MODBUS_INEPRO_RegAddress[i,4]:=16#2020;
MODBUS_INEPRO_RegDescr[i,4]:='Grid frequency';
MODBUS_INEPRO_RegQuantity[i,4]:=2;
MODBUS_INEPRO_RegValueType[i,4]:=VALUE_REAL;

MODBUS_INEPRO_RegAddress[i,5]:=16#2068;
MODBUS_INEPRO_RegDescr[i,5]:='L1 CURRENT';
MODBUS_INEPRO_RegQuantity[i,5]:=2;
MODBUS_INEPRO_RegValueType[i,5]:=VALUE_REAL;

MODBUS_INEPRO_RegAddress[i,6]:=16#206C;
MODBUS_INEPRO_RegDescr[i,6]:='L2 CURRENT';
MODBUS_INEPRO_RegQuantity[i,6]:=2;
MODBUS_INEPRO_RegValueType[i,6]:=VALUE_REAL;

MODBUS_INEPRO_RegAddress[i,7]:=16#2070;
MODBUS_INEPRO_RegDescr[i,7]:='L3 CURRENT';
MODBUS_INEPRO_RegQuantity[i,7]:=2;
MODBUS_INEPRO_RegValueType[i,7]:=VALUE_REAL;

MODBUS_INEPRO_RegAddress[i,8]:=16#2080;
MODBUS_INEPRO_RegDescr[i,8]:='ACTIVE POWER';
MODBUS_INEPRO_RegQuantity[i,8]:=2;
MODBUS_INEPRO_RegValueType[i,8]:=VALUE_REAL;

MODBUS_INEPRO_RegAddress[i,9]:=16#2088;
MODBUS_INEPRO_RegDescr[i,9]:='L1 ACTIVE POWER';
MODBUS_INEPRO_RegQuantity[i,9]:=2;
MODBUS_INEPRO_RegValueType[i,9]:=VALUE_REAL;

MODBUS_INEPRO_RegAddress[i,10]:=16#208C;
MODBUS_INEPRO_RegDescr[i,10]:='L2 ACTIVE POWER';
MODBUS_INEPRO_RegQuantity[i,10]:=2;
MODBUS_INEPRO_RegValueType[i,10]:=VALUE_REAL;

MODBUS_INEPRO_RegAddress[i,11]:=16#2090;
MODBUS_INEPRO_RegDescr[i,11]:='L3 ACTIVE POWER';
MODBUS_INEPRO_RegQuantity[i,11]:=2;
MODBUS_INEPRO_RegValueType[i,11]:=VALUE_REAL;

MODBUS_INEPRO_RegAddress[i,12]:=16#20A0;
MODBUS_INEPRO_RegDescr[i,12]:='REACTIVE POWER';
MODBUS_INEPRO_RegQuantity[i,12]:=2;
MODBUS_INEPRO_RegValueType[i,12]:=VALUE_REAL;

MODBUS_INEPRO_RegAddress[i,13]:=16#20A8;
MODBUS_INEPRO_RegDescr[i,13]:='L1 REACTIVE POWER';
MODBUS_INEPRO_RegQuantity[i,13]:=2;
MODBUS_INEPRO_RegValueType[i,13]:=VALUE_REAL;

MODBUS_INEPRO_RegAddress[i,14]:=16#20AC;
MODBUS_INEPRO_RegDescr[i,14]:='L2 REACTIVE POWER';
MODBUS_INEPRO_RegQuantity[i,14]:=2;
MODBUS_INEPRO_RegValueType[i,14]:=VALUE_REAL;

MODBUS_INEPRO_RegAddress[i,15]:=16#20B0;
MODBUS_INEPRO_RegDescr[i,15]:='L3 REACTIVE POWER';
MODBUS_INEPRO_RegQuantity[i,15]:=2;
MODBUS_INEPRO_RegValueType[i,15]:=VALUE_REAL;

MODBUS_INEPRO_RegAddress[i,16]:=16#20C0;
MODBUS_INEPRO_RegDescr[i,16]:='APPARENT POWER';
MODBUS_INEPRO_RegQuantity[i,16]:=2;
MODBUS_INEPRO_RegValueType[i,16]:=VALUE_REAL;

MODBUS_INEPRO_RegAddress[i,17]:=16#20C8;
MODBUS_INEPRO_RegDescr[i,17]:='L1 APPARENT POWER';
MODBUS_INEPRO_RegQuantity[i,17]:=2;
MODBUS_INEPRO_RegValueType[i,17]:=VALUE_REAL;

MODBUS_INEPRO_RegAddress[i,18]:=16#20CC;
MODBUS_INEPRO_RegDescr[i,18]:='L2 APPARENT POWER';
MODBUS_INEPRO_RegQuantity[i,18]:=2;
MODBUS_INEPRO_RegValueType[i,18]:=VALUE_REAL;

MODBUS_INEPRO_RegAddress[i,19]:=16#20D0;
MODBUS_INEPRO_RegDescr[i,19]:='L3 APPARENT POWER';
MODBUS_INEPRO_RegQuantity[i,19]:=2;
MODBUS_INEPRO_RegValueType[i,19]:=VALUE_REAL;

MODBUS_INEPRO_RegAddress[i,20]:=16#20E0;
MODBUS_INEPRO_RegDescr[i,20]:='POWER FACTOR';
MODBUS_INEPRO_RegQuantity[i,20]:=2;
MODBUS_INEPRO_RegValueType[i,20]:=VALUE_REAL;

MODBUS_INEPRO_RegAddress[i,21]:=16#20E8;
MODBUS_INEPRO_RegDescr[i,21]:='L1 POWER FACTOR';
MODBUS_INEPRO_RegQuantity[i,21]:=2;
MODBUS_INEPRO_RegValueType[i,21]:=VALUE_REAL;

MODBUS_INEPRO_RegAddress[i,22]:=16#20EC;
MODBUS_INEPRO_RegDescr[i,22]:='L2 POWER FACTOR';
MODBUS_INEPRO_RegQuantity[i,22]:=2;
MODBUS_INEPRO_RegValueType[i,22]:=VALUE_REAL;

MODBUS_INEPRO_RegAddress[i,23]:=16#20F0;
MODBUS_INEPRO_RegDescr[i,23]:='L3 POWER FACTOR';
MODBUS_INEPRO_RegQuantity[i,23]:=2;
MODBUS_INEPRO_RegValueType[i,23]:=VALUE_REAL;

MODBUS_INEPRO_RegAddress[i,24]:=16#3000;
MODBUS_INEPRO_RegDescr[i,24]:='TOTAL ACTIVE ENERGY';
MODBUS_INEPRO_RegQuantity[i,24]:=2;
MODBUS_INEPRO_RegValueType[i,24]:=VALUE_REAL;

MODBUS_INEPRO_RegAddress[i,25]:=16#3060;
MODBUS_INEPRO_RegDescr[i,25]:='TOTAL REACTIVE ENERGY';
MODBUS_INEPRO_RegQuantity[i,25]:=2;
MODBUS_INEPRO_RegValueType[i,25]:=VALUE_REAL;

MODBUS_INEPRO_RegAddress[i,26]:=16#1000;
MODBUS_INEPRO_RegDescr[i,26]:='SERIAL_NUMBER';
MODBUS_INEPRO_RegQuantity[i,26]:=2;
MODBUS_INEPRO_RegValueType[i,26]:=VALUE_LONG;

END_FOR
END_FUNCTION

(* POU Utils Functions/AVERAGE_T, ST *)
FUNCTION_BLOCK AVERAGE_T
VAR_INPUT
	IN: 	INT;
END_VAR
VAR_OUTPUT
	HI:		INT;
	AVG:	INT;
	LOW:	INT;
	ERR:	BOOL;
END_VAR
VAR
	sum:	DINT;
	cnt:	WORD;
END_VAR
IF cnt>=65000 THEN
	ERR:=TRUE;
	Read();
	sum := sum - AVG;
	cnt := cnt + 1;
END_IF

sum := sum + IN;
cnt := cnt + 1;

IF IN<LOW THEN  LOW:=IN; END_IF
IF IN>HI  THEN HI :=IN; END_IF
END_FUNCTION_BLOCK
ACTION Read:
AVG := DINT_TO_INT(sum/cnt);
END_ACTION
ACTION Reset:
HI:=IN;
AVG:=IN;
LOW:=IN;
ERR:=FALSE;

sum:=IN;
cnt:=1;
END_ACTION

(* POU ClevergyBlocks/OBJ_ANZ_INEPRO_PRO380/BUILD_REAL_COPY, ST *)
FUNCTION BUILD_REAL_COPY : REAL
VAR_INPUT
		W1	:	WORD;
		W2	:	WORD;
END_VAR
VAR
 	awWords      : ARRAY[1..2] OF WORD;
  	pReal : POINTER TO REAL;
  	rReal : REAL;
END_VAR
awWords[1] := W1;
awWords[2] := W2;
pReal := ADR(awWords);
rReal := pReal^;
BUILD_REAL_COPY:=rReal;
END_FUNCTION

(* POU Utils Functions/COPY_32SWAP16, ST *)
FUNCTION COPY_32SWAP16:BOOL
VAR_INPUT
	pSourceAddress		:POINTER TO ARRAY[1..2] OF WORD;
	pDestinationAddress	:POINTER TO ARRAY[1..2] OF WORD;
END_VAR
VAR
END_VAR
pDestinationAddress^[1]:=pSourceAddress^[2];
pDestinationAddress^[2]:=pSourceAddress^[1];
END_FUNCTION

(* POU Utils Functions/FLT_EVENT, ST *)
FUNCTION_BLOCK FLT_EVENT
VAR_INPUT
	IN		: BOOL;
	INITEV	: BOOL:=TRUE;
END_VAR
VAR_OUTPUT
	EVH		: BOOL;
	EVL		: BOOL;
END_VAR
VAR
	init	: BOOL:=FALSE;
	old		: BOOL;
END_VAR
EVH:=FALSE;
EVL:=FALSE;

IF NOT init THEN
	init:=TRUE;
	IF INITEV THEN
		old := NOT IN;
	ELSE
		old := IN;
	END_IF
END_IF

IF old<>IN THEN
	old:=IN;
	IF IN THEN EVH:=TRUE; ELSE EVL:=TRUE; END_IF
END_IF
END_FUNCTION_BLOCK

(* POU Utils Functions/FLT_TIME, ST *)
FUNCTION_BLOCK FLT_TIME
VAR_INPUT
	IN		: BOOL;
	TTAP	: TIME:=T#5s;
	INITEV	: BOOL:=TRUE;
END_VAR
VAR_OUTPUT
	OUT		: BOOL;
	EVH		: BOOL;
	EVL		: BOOL;
END_VAR
VAR
	init	: BOOL:=FALSE;
	timer	: TON;
END_VAR
EVH:=FALSE;
EVL:=FALSE;

IF NOT init THEN
	init := TRUE;
	IF INITEV THEN
		OUT  := NOT IN;
	ELSE
		OUT  := IN;
	END_IF
END_IF

IF OUT<>IN THEN
	timer(IN:=TRUE,PT:=TTAP);
	IF timer.Q THEN
		OUT:=IN;
		timer(IN:=FALSE);
		IF OUT THEN EVH:=TRUE; ELSE EVL:=TRUE; END_IF
	END_IF
ELSE
	timer(IN:=FALSE);
END_IF
END_FUNCTION_BLOCK

(* POU Utils/FUN_ByteAsci, ST *)
FUNCTION FUN_ByteAsci : STRING(1)
VAR_INPUT
	ByteIn:BYTE;
END_VAR
VAR
END_VAR
CASE ByteIn OF

	32: FUN_ByteAsci:=' ';
	33: FUN_ByteAsci:='!';
	34: FUN_ByteAsci:='"';
	35: FUN_ByteAsci:='#';

	37: FUN_ByteAsci:='%';
	38: FUN_ByteAsci:='&';

	40: FUN_ByteAsci:='(';
	41: FUN_ByteAsci:=')';
	42: FUN_ByteAsci:='*';
	43: FUN_ByteAsci:='+';
	44: FUN_ByteAsci:=',';
	45: FUN_ByteAsci:='-';
	46: FUN_ByteAsci:='.';
	47: FUN_ByteAsci:='/';
	48: FUN_ByteAsci:='0';
	49: FUN_ByteAsci:='1';
	50: FUN_ByteAsci:='2';
	51: FUN_ByteAsci:='3';
	52: FUN_ByteAsci:='4';
	53: FUN_ByteAsci:='5';
	54: FUN_ByteAsci:='6';
	55: FUN_ByteAsci:='7';
	56: FUN_ByteAsci:='8';
	57: FUN_ByteAsci:='9';
	58: FUN_ByteAsci:=':';
	59: FUN_ByteAsci:=';';
	60: FUN_ByteAsci:='<';
	61: FUN_ByteAsci:='=';
	62: FUN_ByteAsci:='>';
	63: FUN_ByteAsci:='?';
	64: FUN_ByteAsci:='@';
	65: FUN_ByteAsci:='A';
	66: FUN_ByteAsci:='B';
	67: FUN_ByteAsci:='C';
	68: FUN_ByteAsci:='D';
	69: FUN_ByteAsci:='E';
	70: FUN_ByteAsci:='F';
	71: FUN_ByteAsci:='G';
	72: FUN_ByteAsci:='H';
	73: FUN_ByteAsci:='I';
	74: FUN_ByteAsci:='J';
	75: FUN_ByteAsci:='K';
	76: FUN_ByteAsci:='L';
	77: FUN_ByteAsci:='M';
	78: FUN_ByteAsci:='N';
	79: FUN_ByteAsci:='O';
	80: FUN_ByteAsci:='P';
	81: FUN_ByteAsci:='Q';
	82: FUN_ByteAsci:='R';
	83: FUN_ByteAsci:='S';
	84: FUN_ByteAsci:='T';
	85: FUN_ByteAsci:='U';
	86: FUN_ByteAsci:='V';
	87: FUN_ByteAsci:='W';
	88: FUN_ByteAsci:='X';
	89: FUN_ByteAsci:='Y';
	90: FUN_ByteAsci:='Z';
	91: FUN_ByteAsci:='[';
	92: FUN_ByteAsci:='\';
	93: FUN_ByteAsci:=']';
	94: FUN_ByteAsci:='^';
	95: FUN_ByteAsci:='_';
	96: FUN_ByteAsci:='`';
	97: FUN_ByteAsci:='a';
	98: FUN_ByteAsci:='b';
	99: FUN_ByteAsci:='c';
	100: FUN_ByteAsci:='d';
	101: FUN_ByteAsci:='e';
	102: FUN_ByteAsci:='f';
	103: FUN_ByteAsci:='g';
	104: FUN_ByteAsci:='h';
	105: FUN_ByteAsci:='i';
	106: FUN_ByteAsci:='j';
	107: FUN_ByteAsci:='k';
	108: FUN_ByteAsci:='l';
	109: FUN_ByteAsci:='m';
	110: FUN_ByteAsci:='n';
	111: FUN_ByteAsci:='o';
	112: FUN_ByteAsci:='p';
	113: FUN_ByteAsci:='q';
	114: FUN_ByteAsci:='r';
	115: FUN_ByteAsci:='s';
	116: FUN_ByteAsci:='t';
	117: FUN_ByteAsci:='u';
	118: FUN_ByteAsci:='v';
	119: FUN_ByteAsci:='w';
	120: FUN_ByteAsci:='x';
	121: FUN_ByteAsci:='y';
	122: FUN_ByteAsci:='z';
	123: FUN_ByteAsci:='{';
	124: FUN_ByteAsci:='|';
	125: FUN_ByteAsci:='}';
	126: FUN_ByteAsci:='~';

	167: FUN_ByteAsci:='°';
	176: FUN_ByteAsci:='°';


ELSE
	FUN_ByteAsci:='';

END_CASE
END_FUNCTION

(* POU Utils Functions/LAMP_AL_GENERALE, ST *)
FUNCTION_BLOCK LAMP_AL_GENERALE
VAR_INPUT

	Allarme: BOOL;
	Warning: BOOL;
END_VAR
VAR_OUTPUT
	SistemaOK:BOOL;
	SistemaInAllarme:BOOL;
	SistemaWarning:BOOL;
	AllarmeLampada:BOOL;
END_VAR
VAR
	Lampeggio:BLINK;
END_VAR
IF Allarme THEN       					(* Se Allarme Attivo Lucde fissa ON *)
	SistemaInAllarme:=TRUE;
	SistemaWarning:=FALSE;
	AllarmeLampada:=TRUE;
ELSIF Warning THEN					(* Se Allarme Attivo Lucde fissa pulse *)
	SistemaInAllarme:=FALSE;
	SistemaWarning:=TRUE;
	Lampeggio(ENABLE:=TRUE , TIMELOW:=t#1s , TIMEHIGH:=t#1s , OUT=>AllarmeLampada );
ELSE
	SistemaInAllarme:=FALSE;
	SistemaWarning:=FALSE;
	AllarmeLampada:=FALSE;
END_IF
END_FUNCTION_BLOCK

(* POU Utils Functions/LINEAR_BAD, ST *)
FUNCTION LINEAR_BAD : INT (* Linear interpolation *)
VAR_INPUT
	PuntoMinX	: INT;
	PuntoMaxX	: INT;
	ValIn		: INT;
	PuntoMinY	: REAL;
	PuntoMaxY	: REAL;
	Decimali	: BYTE;
END_VAR
VAR
	Gain				: REAL;
	PuntoMinX_R			: REAL;
	PuntoMaxX_R			: REAL;
	Linearizzazione_R	: REAL;
END_VAR
PuntoMinX_R:=INT_TO_REAL(PuntoMinX);
PuntoMaxX_R:=INT_TO_REAL(PuntoMaxX);

Gain:=(PuntoMaxX_R-PuntoMinX_R)/(PuntoMaxY-PuntoMinY);	(* Calcolo in guadagno per la linarizzazione *)
Linearizzazione_R:=PuntoMinx+(Gain*(ValIn-PuntoMinY));	(* Ottengo il valore linearizzato *)

LINEAR_BAD:=REAL_TO_INT(Linearizzazione_R*(EXPT(10, Decimali)));  (* Ottengo intero con i decimai voluti *)
END_FUNCTION

(* POU TCP_Logger/LogTrig, ST *)
FUNCTION LogTrig : BOOL
VAR
	s1 : STRING(160);
	i  : BYTE;
	j  : WORD;
END_VAR
(*---------------------------------------------------------------*)
	Logger_Head();
(*---------------------------------------------------------------*)

PX01.AddLogData();
PX02.AddLogData();
PX03.AddLogData();
PX04.AddLogData();
Logger_Send();


Logger_Head();

(*
FOR i:=1 TO Plant_ANZ_INEPRO DO
	ANZ_INEPRO[i].AddLogData();
END_FOR *)
ANZ_INEPRO[1].AddLogData();
ANZ_INEPRO[2].AddLogData();
Logger_Send();


Logger_Head();

ANZ_INEPRO[3].AddLogData();
ANZ_INEPRO[4].AddLogData();
Logger_Send();


Logger_Head();
ANZ_INEPRO[5].AddLogData();

Logger_Send();


Logger_Head();

	COMPRESSORE01.AddLogData(ModBus:=MODB02);
	COMPRESSORE05.AddLogData(ModBus:=MODB02);
Logger_Send();


Logger_Head();
	COMPRESSORE02.AddLogData(ModBus:=MODB03);
	COMPRESSORE03.AddLogData(ModBus:=MODB03);
	COMPRESSORE04.AddLogData(ModBus:=MODB03);
Logger_Send();


Logger_Head();

	FPT01.AddLogData(ModBus:=MODB05);
	FPT02.AddLogData();
	FPT03.AddLogData();
	FPT04.AddLogData();
	FPT05.AddLogData();
	FPT06.AddLogData();
	FPT07.AddLogData();
	FPT08.AddLogData();
	FPT09.AddLogData();
	FPT10.AddLogData();

(*	ESSICATORE01.AddLogData(ModBus:=MODB04); *)
(*	ESSICATORE02.AddLogData(ModBus:=MODB04); *)



(*---------------------------------------------------------------*)
	Logger_Send();
(*---------------------------------------------------------------*)
END_FUNCTION

(* POU Utils Functions/MEMCLR, ST *)
FUNCTION MEMCLR:BOOL
VAR_INPUT
	pDestinationAddress:POINTER TO ARRAY[1..2] OF BYTE;
	BytesToClear:WORD;
END_VAR
VAR
END_VAR
WHILE (BytesToClear > 0) DO
	pDestinationAddress^[1]:=0;
	pDestinationAddress:=ADR(pDestinationAddress^[2]); (* increment destination *)
	BytesToClear:=BytesToClear -1; (* decrement number of bytes to copy *)
END_WHILE
END_FUNCTION

(* POU Plant_Objects/obj_AI_GEN, ST *)
FUNCTION_BLOCK obj_AI_GEN
(* === TEMPERATURE PROBE FROM ANALOG INPUT ===
   v1.0[16/04/05] - Versioning
*)
VAR_INPUT
	(* Settings *)
	ID				: BYTE;
	PuntoMinX		: INT;			(* Parametri per la scalatura *)
	PuntoMaxX		: INT;
	PuntoMinY		: REAL;
	PuntoMaxY		: REAL;
	Decimali		: BYTE:=1;
	SogliaHH		: WORD;			(* Soglia per segnalazione Allarme Extra Range in alto - Solitamente sondo in CC *)
	SogliaHL		: WORD;			(* Soglia per segnalazione Allarme Extra Range in Basso - Solitamente sondo Aperta *)
	SogliaWH		: REAL;			(* Soglia per segnalazione Warning  in alto  *)
	SogliaWL		: REAL;    		(* Soglia per segnalazione Warning in basso  *)
	TAP				: INT:=2000;	(* Filtro in msec *)
	INITEV			: BOOL:= TRUE;	(* Generate init OK event *)
	(* Physical input *)
	AI_INPUT		: WORD;    		(* Sensor analog input *)
	TipoSensore:STRING(12);
END_VAR
VAR_OUTPUT
	WRN				: BOOL;	(* Segnalazione Warning *)
	ERR				: BOOL; (* Segnalazione Errore *)
	ValoreScalato	: INT;
	(* Status *)
	Status_Log	: BYTE;
	Status_Vis 	: DWORD;
END_VAR
VAR
	SegnaleHH	: BOOL;
	SegnaleHL	: BOOL;
	SegnaleOK	: BOOL;
	SegnaleWH	: BOOL;
	SegnaleWL	: BOOL;
    FiltroWRN	: TON;
    FiltroOK	: TON;
    FiltroERR	: TON;
END_VAR
(* Verifico che le variabile letta dall'ingresso Analogico  sia dentro i range
ATTENZIONE I LIMITI SPESSO SONO IN WORD VERIFICA  TABELLA MANUALE WAGO  *)

SegnaleHH:=(AI_INPUT>=SogliaHH);
SegnaleHL:=(AI_INPUT<=SogliaHL);
SegnaleOK:=NOT (SegnaleHH OR SegnaleHL);

(* Linerarizzo il segnale di ingresso e la converto in unita ingegneristiche *)
ValoreScalato:=LINEAR_BAD(PuntoMinX, PuntoMaxX, AI_INPUT, PuntoMinY, PuntoMaxY, Decimali);


IF SegnaleOK  THEN
	(*  Verifica  e segnalazione Warning *)
	SegnaleWH:=(ValoreScalato>SogliaWH*(EXPT(10, Decimali)));
	SegnaleWL:=(ValoreScalato<SogliaWL*(EXPT(10, Decimali)));

	Status_Log:=0;
	Status_Vis:=16#20F020;    (* Indicazione WEB Visu Sonda OK *)

	FiltroWRN( IN:=(SegnaleWH OR SegnaleWL), PT:=INT_TO_TIME(TAP) );    (* Filtro su LOG *)
	IF  FiltroWRN.Q THEN     (* Condizione di WARNING *)
		IF NOT WRN THEN
			WRN:=TRUE;
			Status_Log:=1;
			LogEv(EL_Wrn,EO_TPV,ID,SEL(ValoreScalato<=SogliaWL,3,2),INT_TO_STRING(ValoreScalato));
		END_IF
	END_IF

    IF (INITEV OR WRN OR ERR) AND NOT FiltroWRN.Q THEN
		FiltroWRN(IN:=FALSE  , PT:=INT_TO_TIME(TAP));    (* Resetto il Filtro su LOG WRN  *)
		FiltroERR(IN:=FALSE  , PT:=INT_TO_TIME(TAP));    (* Resetto il Filtro su LOG ERR *)
		INITEV:=FALSE; ERR:=FALSE; WRN:=FALSE;
		LogEv(EL_Log,EO_TPV,ID,1,'');
	END_IF
ELSE
	FiltroERR(IN:=TRUE  , PT:= INT_TO_TIME(TAP) );    (* Filtro su LOG *)
	IF  FiltroERR.Q THEN     (* Condizione di WARNING *)
		IF NOT ERR THEN
			ERR:=TRUE;
			Status_Log:=2;

			IF SegnaleHH THEN LogEv(EL_Alarm,EO_TPV,ID,6,INT_TO_STRING(ValoreScalato));END_IF;
			IF SegnaleHL THEN LogEv(EL_Alarm,EO_TPV,ID,4,INT_TO_STRING(ValoreScalato));END_IF;
		END_IF
	END_IF

	Status_Vis:=16#2020F0;   (* Indicazione WEB Visu Sonda KO *)
END_IF



(* Status Log *)
IF ERR THEN
	Status_Log := 2;
	Status_Vis := COLOR_RED;
ELSIF WRN THEN
	Status_Log := 1;
	Status_Vis := COLOR_YELLOW;
ELSE
	Status_Log := 0; Status_Vis := COLOR_GREEN;
END_IF
END_FUNCTION_BLOCK
ACTION AddLogData:
Logger.s1:=CONCAT('&',TipoSensore);
IF ID<10 THEN Logger.s1:=CONCAT(Logger.s1,'0');END_IF
Logger.s1:=CONCAT(Logger.s1,BYTE_TO_STRING(ID));
Logger.s1:=CONCAT(Logger.s1,'=');


Logger.s1:=CONCAT(Logger.s1,WORD_TO_STRING(Status_Log));		Logger.s1:=CONCAT(Logger.s1,';');
Logger.s1:=CONCAT(Logger.s1,INT_TO_STRING(ValoreScalato));


ADDSTRING(ADR(Logger.TData), ADR(Logger.s1), Logger.TLen);
END_ACTION

(* POU ClevergyBlocks/OBJ_ANZ_INEPRO_PRO380/obj_ANZ_INEPRO_PRO380, ST *)
FUNCTION_BLOCK obj_ANZ_INEPRO_PRO380
(* === Block for realizing the ANZ entity with the meter INEPRO PRO380 ===
	
	One ANZ block manages one physical ANZ device.
	
	Versioning:
		v1.0 [28/07/16] - Diego Bernini
*)
VAR_INPUT

	(* Logical ID of the ANZ, univocal w.r.t the plant *)
	ID										 : WORD;
	(* Type of ANZ: 1-phase or 3-phase *)
	contabilizerMode							 : en_ANZ_Type := THREE_PHASE;

	modbusConnector: obj_MODBUS_GENERIC_CONNECTOR;

	(* meter dependent fields, by the connector*)
	specificData								:  typ_ANZ_INEPRO_PRO380;

	(* determines if warning errors are sent or not *)
	enableWarning : BOOL :=FALSE;

	TIMING_AGGREGATED_MEASURE:TIME;
	TIMING_RESET_AGGREGATED_MEASURE:TIME;

END_VAR

VAR_OUTPUT

	(* output records representing the data in according to the ANZ Clevergy Web format *)
	measures						: typ_ANZ_real;
	(*status of the block according the Clevergy architecture *)
	Status_Log						: BYTE;
	Status_Vis	:	DWORD;

END_VAR

VAR

	contAvg								 : REAL :=0;
	sumAvg								 : REAL :=0;
	timerCalc								 : TON;
	timerReset							 : TON;

	alarmMsg : STRING;
	alarmLaunched: ARRAY[1..MAX_ALARM] OF BYTE;

	warningMsg : STRING;
	warningLaunched: ARRAY[1..MAX_WARNING] OF BYTE;

	i : BYTE;
	tmpAlarm:BYTE;
	tmpWarning:BYTE;

END_VAR
VAR CONSTANT
	MAX_ALARM :BYTE:=20;
	MAX_WARNING :BYTE:=20;
END_VAR
VAR
	CheckEvents: BOOL;
END_VAR
Status_Log:=ModBusConnector.Status_Log;

getModbusData();

timerReset(IN:=NOT timerReset.Q,PT:=TIMING_RESET_AGGREGATED_MEASURE);
IF timerReset.Q THEN

	sumAvg := 0;
	contAvg := 0;

 	specificData.rMaximumTotalActivePower:=0; (* reset => min possible val *)
	specificData.rMaximumTotalReactivePower:= -2147483648;
	specificData.rMaximumCurrentL1:=0;
	specificData.rMaximumCurrentL2:=0;
	specificData.rMaximumCurrentL3:=0;

END_IF

(*compute additional measures, the ones which are not provided directly*)
timerCalc(IN:=NOT timerCalc.Q,PT:=TIMING_AGGREGATED_MEASURE);

IF timerCalc.Q THEN
	sumAvg := sumAvg+specificData.rTotalActivePower;
	contAvg:=contAvg+1;
	specificData.rAverageTotalActivePower:=sumAvg/contAvg;
	IF specificData.rTotalActivePower > specificData.rMaximumTotalActivePower THEN specificData.rMaximumTotalActivePower:= specificData.rTotalActivePower; END_IF
	IF specificData.rTotalReactivePower > specificData.rMaximumTotalReactivePower THEN specificData.rMaximumTotalReactivePower:= specificData.rTotalReactivePower; END_IF

	IF specificData.arCurrent[1] > specificData.rMaximumCurrentL1 THEN specificData.rMaximumCurrentL1:= specificData.arCurrent[1]; END_IF
	IF specificData.arCurrent[2] > specificData.rMaximumCurrentL2 THEN specificData.rMaximumCurrentL2:= specificData.arCurrent[2]; END_IF
	IF specificData.arCurrent[3] > specificData.rMaximumCurrentL3 THEN specificData.rMaximumCurrentL3:= specificData.arCurrent[3]; END_IF

END_IF


(* convert the data to the Clevergy format *)
convertToClevergyFormat();

(* visu	*)
IF Status_Log = 2 THEN
	Status_Vis := COLOR_RED;
ELSIF Status_Log = 1 THEN
	Status_Vis := COLOR_YELLOW;
ELSE
	Status_Vis := COLOR_GREEN;
END_IF
END_FUNCTION_BLOCK
ACTION AddLogData:
Logger.s1:=INSERT('&ANZ=',WORD_TO_STRING(ID),4);
IF ID<10 THEN Logger.s1:=INSERT(Logger.s1,'0',4); END_IF

Logger.s1:=CONCAT(Logger.s1,REAL_TO_STRING(measures.V_L1N));		Logger.s1:=CONCAT(Logger.s1,';');
Logger.s1:=CONCAT(Logger.s1,REAL_TO_STRING(measures.V_L2N));		Logger.s1:=CONCAT(Logger.s1,';');
Logger.s1:=CONCAT(Logger.s1,REAL_TO_STRING(measures.V_L3N));		Logger.s1:=CONCAT(Logger.s1,';');
Logger.s1:=CONCAT(Logger.s1,REAL_TO_STRING(measures.V_L1L2));		Logger.s1:=CONCAT(Logger.s1,';');
Logger.s1:=CONCAT(Logger.s1,REAL_TO_STRING(measures.V_L2L3));		Logger.s1:=CONCAT(Logger.s1,';');
Logger.s1:=CONCAT(Logger.s1,REAL_TO_STRING(measures.V_L3L1));		Logger.s1:=CONCAT(Logger.s1,';');

Logger.s1:=CONCAT(Logger.s1,REAL_TO_STRING(measures.FREQ));		Logger.s1:=CONCAT(Logger.s1,';');

Logger.s1:=CONCAT(Logger.s1,REAL_TO_STRING(measures.I_L1));		Logger.s1:=CONCAT(Logger.s1,';');
Logger.s1:=CONCAT(Logger.s1,REAL_TO_STRING(measures.I_L2));		Logger.s1:=CONCAT(Logger.s1,';');
Logger.s1:=CONCAT(Logger.s1,REAL_TO_STRING(measures.I_L3));		Logger.s1:=CONCAT(Logger.s1,';');
Logger.s1:=CONCAT(Logger.s1,REAL_TO_STRING(measures.I_L1_Max)); 	Logger.s1:=CONCAT(Logger.s1,';');
Logger.s1:=CONCAT(Logger.s1,REAL_TO_STRING(measures.I_L2_Max)); 	Logger.s1:=CONCAT(Logger.s1,';');
Logger.s1:=CONCAT(Logger.s1,REAL_TO_STRING(measures.I_L3_Max)); 	Logger.s1:=CONCAT(Logger.s1,';');

Logger.s1:=CONCAT(Logger.s1,REAL_TO_STRING(measures.PF_L1));		Logger.s1:=CONCAT(Logger.s1,';');
Logger.s1:=CONCAT(Logger.s1,REAL_TO_STRING(measures.PF_L2));		Logger.s1:=CONCAT(Logger.s1,';');
Logger.s1:=CONCAT(Logger.s1,REAL_TO_STRING(measures.PF_L3));		Logger.s1:=CONCAT(Logger.s1,';');

Logger.s1:=CONCAT(Logger.s1,REAL_TO_STRING(measures.P_3P));		Logger.s1:=CONCAT(Logger.s1,';');
Logger.s1:=CONCAT(Logger.s1,REAL_TO_STRING(measures.P_3P_Avg)); 	Logger.s1:=CONCAT(Logger.s1,';');
Logger.s1:=CONCAT(Logger.s1,REAL_TO_STRING(measures.P_3P_Max)); 	Logger.s1:=CONCAT(Logger.s1,';');

Logger.s1:=CONCAT(Logger.s1,REAL_TO_STRING(measures.Q_3P));			Logger.s1:=CONCAT(Logger.s1,';');
Logger.s1:=CONCAT(Logger.s1, REAL_TO_STRING(measures.Q_3P_Max));		Logger.s1:=CONCAT(Logger.s1,';');

Logger.s1:=CONCAT(Logger.s1,REAL_TO_STRING(measures.WH_3P));			Logger.s1:=CONCAT(Logger.s1,';');
Logger.s1:=CONCAT(Logger.s1,REAL_TO_STRING(measures.VARH_3P));			Logger.s1:=CONCAT(Logger.s1,';');

Logger.s1:=CONCAT(Logger.s1,BYTE_TO_STRING(Status_Log)); 					Logger.s1:=CONCAT(Logger.s1,';');

Logger.s1:=CONCAT(Logger.s1,REAL_TO_STRING(measures.COSPHI_L1));		Logger.s1:=CONCAT(Logger.s1,';');
Logger.s1:=CONCAT(Logger.s1,REAL_TO_STRING(measures.COSPHI_L2));		Logger.s1:=CONCAT(Logger.s1,';');
Logger.s1:=CONCAT(Logger.s1,REAL_TO_STRING(measures.COSPHI_L3));		Logger.s1:=CONCAT(Logger.s1,';');

Logger.s1:=CONCAT(Logger.s1,BYTE_TO_STRING(SEL(contabilizerMode=THREE_PHASE,1,0)));

ADDSTRING(ADR(Logger.TData), ADR(Logger.s1), Logger.TLen);
END_ACTION
ACTION AddLogData_OLD:
(*Logger.s1:=INSERT('&ANZ=',WORD_TO_STRING(ID),4);
IF ID<10 THEN Logger.s1:=INSERT(Logger.s1,'0',4); END_IF

Logger.s1:=CONCAT(Logger.s1,DWORD_TO_STRING(measures.V_L1N));		Logger.s1:=CONCAT(Logger.s1,';');
Logger.s1:=CONCAT(Logger.s1,DWORD_TO_STRING(measures.V_L2N));		Logger.s1:=CONCAT(Logger.s1,';');
Logger.s1:=CONCAT(Logger.s1,DWORD_TO_STRING(measures.V_L3N));		Logger.s1:=CONCAT(Logger.s1,';');
Logger.s1:=CONCAT(Logger.s1,DWORD_TO_STRING(measures.V_L1L2));		Logger.s1:=CONCAT(Logger.s1,';');
Logger.s1:=CONCAT(Logger.s1,DWORD_TO_STRING(measures.V_L2L3));		Logger.s1:=CONCAT(Logger.s1,';');
Logger.s1:=CONCAT(Logger.s1,DWORD_TO_STRING(measures.V_L3L1));		Logger.s1:=CONCAT(Logger.s1,';');

Logger.s1:=CONCAT(Logger.s1,DWORD_TO_STRING(measures.FREQ));		Logger.s1:=CONCAT(Logger.s1,';');

Logger.s1:=CONCAT(Logger.s1,DWORD_TO_STRING(measures.I_L1));		Logger.s1:=CONCAT(Logger.s1,';');
Logger.s1:=CONCAT(Logger.s1,DWORD_TO_STRING(measures.I_L2));		Logger.s1:=CONCAT(Logger.s1,';');
Logger.s1:=CONCAT(Logger.s1,DWORD_TO_STRING(measures.I_L3));		Logger.s1:=CONCAT(Logger.s1,';');
Logger.s1:=CONCAT(Logger.s1,DWORD_TO_STRING(measures.I_L1_Max)); 	Logger.s1:=CONCAT(Logger.s1,';');
Logger.s1:=CONCAT(Logger.s1,DWORD_TO_STRING(measures.I_L2_Max)); 	Logger.s1:=CONCAT(Logger.s1,';');
Logger.s1:=CONCAT(Logger.s1,DWORD_TO_STRING(measures.I_L3_Max)); 	Logger.s1:=CONCAT(Logger.s1,';');

Logger.s1:=CONCAT(Logger.s1,DINT_TO_STRING(measures.PF_L1));		Logger.s1:=CONCAT(Logger.s1,';');
Logger.s1:=CONCAT(Logger.s1,DINT_TO_STRING(measures.PF_L2));		Logger.s1:=CONCAT(Logger.s1,';');
Logger.s1:=CONCAT(Logger.s1,DINT_TO_STRING(measures.PF_L3));		Logger.s1:=CONCAT(Logger.s1,';');

Logger.s1:=CONCAT(Logger.s1,DINT_TO_STRING(measures.P_3P));		Logger.s1:=CONCAT(Logger.s1,';');
Logger.s1:=CONCAT(Logger.s1,DINT_TO_STRING(measures.P_3P_Avg)); 	Logger.s1:=CONCAT(Logger.s1,';');
Logger.s1:=CONCAT(Logger.s1,DINT_TO_STRING(measures.P_3P_Max)); 	Logger.s1:=CONCAT(Logger.s1,';');

Logger.s1:=CONCAT(Logger.s1,DINT_TO_STRING(measures.Q_3P));			Logger.s1:=CONCAT(Logger.s1,';');
Logger.s1:=CONCAT(Logger.s1,DINT_TO_STRING(measures.Q_3P_Max));		Logger.s1:=CONCAT(Logger.s1,';');

Logger.s1:=CONCAT(Logger.s1,DWORD_TO_STRING(measures.WH_3P));			Logger.s1:=CONCAT(Logger.s1,';');
Logger.s1:=CONCAT(Logger.s1,DINT_TO_STRING(measures.VARH_3P));			Logger.s1:=CONCAT(Logger.s1,';');

Logger.s1:=CONCAT(Logger.s1,BYTE_TO_STRING(Status_Log)); 					Logger.s1:=CONCAT(Logger.s1,';');

Logger.s1:=CONCAT(Logger.s1,DINT_TO_STRING(measures.COSPHI_L1));		Logger.s1:=CONCAT(Logger.s1,';');
Logger.s1:=CONCAT(Logger.s1,DINT_TO_STRING(measures.COSPHI_L2));		Logger.s1:=CONCAT(Logger.s1,';');
Logger.s1:=CONCAT(Logger.s1,DINT_TO_STRING(measures.COSPHI_L3));		Logger.s1:=CONCAT(Logger.s1,';');

Logger.s1:=CONCAT(Logger.s1,BYTE_TO_STRING(SEL(contabilizerMode=THREE_PHASE,1,0)));

ADDSTRING(ADR(Logger.TData), ADR(Logger.s1), Logger.TLen);*)
;
END_ACTION
ACTION checkAlarm:
(*IF(alarmLaunched[1]=0 AND typ_750_494_State.xPhase1_OverCurrentSystem) THEN
	alarmLaunched[1]:=2;
	LogEv(EL_Alarm,EO_ANZ,ID,3, 'xPhase1_OverCurrentSystem');
ELSIF (alarmLaunched[1]=2 AND NOT(typ_750_494_State.xPhase1_OverCurrentSystem) ) THEN
	alarmLaunched[1]:=0;
	LogEv(EL_Log,EO_ANZ,ID,4,'xPhase1_OverCurrentSystem');
END_IF*)

;
END_ACTION
ACTION checkEventsToSignal:
CheckAlarm();
CheckWarning();
CheckStatus();
END_ACTION
ACTION checkStatus:
(*tmpAlarm:=0;
FOR I:=1 TO MAX_alarm DO tmpAlarm:=tmpAlarm+alarmLaunched[i]; END_FOR
IF(tmpAlarm>0) THEN status_Log:=2; END_IF

tmpWarning:=0;
FOR I:=1 TO MAX_WARNING DO tmpWarning:=tmpWarning+warningLaunched[i]; END_FOR
IF(status=0 AND tmpWarning>0) THEN status:=1; END_IF

IF (tmpAlarm =0 AND tmpWarning =0) THEN status:=0; END_IF*)
;
END_ACTION
ACTION checkWarning:
IF(enableWarning = FALSE) THEN RETURN; END_IF

(*IF( warningLaunched[1]=0 AND typ_750_494_State.xGeneralError) THEN
	warningLaunched[1]:=2;
	LogEv(EL_Wrn,EO_ANZ,ID,5, 'xGeneralError');
ELSIF (warningLaunched[1]=2 AND NOT(typ_750_494_State.xGeneralError) ) THEN
	warningLaunched[1]:=0;
	LogEv(EL_Log,EO_ANZ,ID,5,'xGeneralError');
END_IF*)

;
END_ACTION
ACTION convertToClevergyFormat:
	measures.V_L1N := specificData.arVoltage_L_N[1];
	measures.V_L2N := specificData.arVoltage_L_N[2];
	measures.V_L3N := specificData.arVoltage_L_N[3];

	(*n/a*)
	measures.V_L1L2:=0;
	measures.V_L2L3:=0;
	measures.V_L3L1:=0;

	measures.FREQ := specificData.arFrequency*1000;

	measures.I_L1 := specificData.arCurrent[1]*1000;
	measures.I_L2 := specificData.arCurrent[2]*1000;
	measures.I_L3 :=specificData.arCurrent[3]*1000;

	measures.I_L1_Max := specificData.rMaximumCurrentL1*1000;
	measures.I_L2_Max := specificData.rMaximumCurrentL2*1000;
	measures.I_L3_Max := specificData.rMaximumCurrentL3*1000;

	measures.PF_L1 := specificData.arPowerFactorPF[1]*1000;
	measures.PF_L2 := specificData.arPowerFactorPF[2]*1000;
	measures.PF_L3 := specificData.arPowerFactorPF[3]*1000;

	measures.P_3P := specificData.rTotalActivePower*1000;
	measures.P_3P_Avg:=specificData.rAverageTotalActivePower*1000;
	measures.P_3P_Max:=specificData.rMaximumTotalActivePower*1000;

	measures.Q_3P:=specificData.rTotalReactivePower*1000;
	measures.Q_3P_Max:=specificData.rMaximumTotalReactivePower*1000;

	measures.WH_3P:=specificData.rTotalActiveEnergy*10;
	measures.VARH_3P:=specificData.rTotalReactiveEnergy*10;

	(*n/a*)
	measures.COSPHI_L1:=0;
	measures.COSPHI_L2:=0;
	measures.COSPHI_L3:=0;
END_ACTION
ACTION convertToClevergyFormat_OLD:
	measures.V_L1N := REAL_TO_DWORD(specificData.arVoltage_L_N[1]);
	measures.V_L2N := REAL_TO_DWORD(specificData.arVoltage_L_N[2]);
	measures.V_L3N := REAL_TO_DWORD(specificData.arVoltage_L_N[3]);

	(*n/a*)
	measures.V_L1L2:=REAL_TO_DWORD(0);
	measures.V_L2L3:=REAL_TO_DWORD(0);
	measures.V_L3L1:=REAL_TO_DWORD(0);

	measures.FREQ := REAL_TO_DWORD(specificData.arFrequency*1000);

	measures.I_L1 := REAL_TO_DWORD(specificData.arCurrent[1]*1000);
	measures.I_L2 := REAL_TO_DWORD(specificData.arCurrent[2]*1000);
	measures.I_L3 := REAL_TO_DWORD(specificData.arCurrent[3]*1000);

	measures.I_L1_Max := REAL_TO_DWORD(specificData.rMaximumCurrentL1*1000);
	measures.I_L2_Max := REAL_TO_DWORD(specificData.rMaximumCurrentL2*1000);
	measures.I_L3_Max := REAL_TO_DWORD(specificData.rMaximumCurrentL3*1000);

	measures.PF_L1 := REAL_TO_DINT(specificData.arPowerFactorPF[1]*1000);
	measures.PF_L2 := REAL_TO_DINT(specificData.arPowerFactorPF[2]*1000);
	measures.PF_L3 := REAL_TO_DINT(specificData.arPowerFactorPF[3]*1000);

	measures.P_3P := REAL_TO_DINT(specificData.rTotalActivePower);
	measures.P_3P_Avg:=REAL_TO_DINT(specificData.rAverageTotalActivePower);
	measures.P_3P_Max:=REAL_TO_DINT(specificData.rMaximumTotalActivePower);

	measures.Q_3P:=REAL_TO_DINT(specificData.rTotalReactivePower);
	measures.Q_3P_Max:=REAL_TO_DINT(specificData.rMaximumTotalReactivePower);

	measures.WH_3P:=REAL_TO_DINT(specificData.rTotalActiveEnergy*10);
	measures.VARH_3P:=REAL_TO_DINT(specificData.rTotalReactiveEnergy*10);

	(*n/a*)
	measures.COSPHI_L1:=REAL_TO_DINT(0);
	measures.COSPHI_L2:=REAL_TO_DINT(0);
	measures.COSPHI_L3:=REAL_TO_DINT(0);
;
END_ACTION
ACTION getModbusData:
specificData.arFrequency:=modBusConnector.regData[4];

specificData.arVoltage_L_N[1]:=modBusConnector.regData[1];
specificData.arVoltage_L_N[2]:=modBusConnector.regData[2];
specificData.arVoltage_L_N[3]:=modBusConnector.regData[3];

specificData.arCurrent[1]:=modBusConnector.regData[5];
specificData.arCurrent[2]:=modBusConnector.regData[6];
specificData.arCurrent[3]:=modBusConnector.regData[7];

specificData.rTotalActivePower:=modBusConnector.regData[8];
specificData.arActivePower[1]:=modBusConnector.regData[9];
specificData.arActivePower[2]:=modBusConnector.regData[10];
specificData.arActivePower[3]:=modBusConnector.regData[11];

specificData.rTotalReactivePower:=modBusConnector.regData[12];
specificData.arReactivePower[1]:=modBusConnector.regData[13];
specificData.arReactivePower[2]:=modBusConnector.regData[14];
specificData.arReactivePower[3]:=modBusConnector.regData[15];

specificData.rTotalApparentPower:=modBusConnector.regData[16];
specificData.arApparentPower[1]:=modBusConnector.regData[17];
specificData.arApparentPower[2]:=modBusConnector.regData[18];
specificData.arApparentPower[3]:=modBusConnector.regData[19];

specificData.rTotalPowerFactorPF:=modBusConnector.regData[20];
specificData.arPowerFactorPF[1]:=modBusConnector.regData[21];
specificData.arPowerFactorPF[2]:=modBusConnector.regData[22];
specificData.arPowerFactorPF[3]:=modBusConnector.regData[23];

specificData.rTotalActiveEnergy:=modBusConnector.regData[24];

specificData.rTotalReactiveEnergy:=modBusConnector.regData[25];
END_ACTION

(* POU ClevergyBlocks/OBJ_ANZ_INEPRO_PRO380/obj_MODBUS_GENERIC_CONNECTOR, ST *)
FUNCTION_BLOCK obj_MODBUS_GENERIC_CONNECTOR
VAR CONSTANT
		(* States of normal modbus data reading *)
		WAIT_STATE			:	BYTE := 0;
		QUERY_START_CYCLE	: 	BYTE := 1;
		QUERY_MEAS_REQ		:  	BYTE := 2;
		QUERY_MEAS_ANSW	: 	BYTE := 3;
		ERROR_STATE			:	BYTE := 4;
END_VAR
VAR_INPUT
		PARENT_EO_TYPE 		: 	WORD;
		PARENT_EO_ID		:	BYTE;
		Address				:	BYTE;
		TIMING				:	TIME:=t#500ms;

		retryErrMax			:	BYTE := 10;

END_VAR
VAR_IN_OUT
		ModBus		:	obj_MODBUS_ANZ;
END_VAR
VAR_OUTPUT
		Status_Log	:	BYTE;
		Status_Vis	:	DWORD;

		regDescr : ARRAY[1..MODBUS_INEPRO_MAX_REG] OF STRING(20);
		regAddress : ARRAY[1..MODBUS_INEPRO_MAX_REG] OF WORD;
		regQuantity : ARRAY[1..MODBUS_INEPRO_MAX_REG] OF BYTE;
		regValueType : ARRAY[1..MODBUS_INEPRO_MAX_REG] OF en_Modbus_Reg_Type;
		regData: ARRAY[1..MODBUS_INEPRO_MAX_REG] OF REAL;
		regDataWord: ARRAY[1..MODBUS_INEPRO_MAX_REG, 1..2] OF WORD;

END_VAR
VAR
		InitOK		:	BOOL := FALSE;

		(* Modbus State machine variables	*)
		state		:	BYTE;
		last_state		:	BYTE;
		retry		:	BYTE;
		retryErr		:	BYTE;
		ReadTmr		:	TON := (PT:=t#5s);	(* Just to do a first ModBus read at the beginning *)
		fModbusAlr	:	BOOL;

		(* Event check variable	*)
		Alarm		:	FLT_EVENT;
		ModBusAlr	:	FLT_EVENT := (INITEV:=FALSE);
		StatusOK		:	FLT_EVENT := (INITEV:=FALSE);
		AlarmCtr		:	BYTE;
		WarningCtr	:	BYTE;

		fTimeout	:	BOOL;

		currentReg:INT:=1;

		i:INT;
		x:INT;
END_VAR
IF NOT InitOK THEN
	ReadTmr.PT := timing;
	InitOK := TRUE;
	initMapping();
END_IF

(* State machine *)
Stm();

(* Check if an alarm has occured *)
CheckAlarm();

(* Set "Status_Log" according to actual object status	*)
IF AlarmCtr > 0 THEN
	Status_Log := 2;
	Status_Vis := COLOR_RED;
ELSIF WarningCtr > 0 THEN
	Status_Log := 1;
	Status_Vis := COLOR_YELLOW;
ELSE
	Status_Log := 0;

	Status_Vis := COLOR_GREEN;
END_IF
END_FUNCTION_BLOCK
ACTION CheckAlarm:
(*** Verify ModBus error	***)
ModbusAlr(IN:=fModbusAlr);

IF ModbusAlr.EVH THEN
	LogEv(EL_Alarm,PARENT_EO_TYPE,PARENT_EO_ID,2,SEL(ModBus.MB_MASTER.MB_Error<>0,'0','1'));
	AlarmCtr := AlarmCtr + 1;
END_IF

IF ModbusAlr.EVL THEN
	LogEv(EL_Log,PARENT_EO_TYPE,PARENT_EO_ID,1,'');
	AlarmCtr := SEL(AlarmCtr=0, AlarmCtr-1, 0);
END_IF
END_ACTION
ACTION initMapping:
FOR I:=1 TO MODBUS_INEPRO_MAX_REG DO

	IF MODBUS_INEPRO_RegAddress[PARENT_EO_ID,i] <> 0 THEN

		regAddress[i]:=MODBUS_INEPRO_RegAddress[PARENT_EO_ID, i];
		REGDescr[i]:=MODBUS_INEPRO_REGDescr[PARENT_EO_ID, i];
		regQuantity[i]:=MODBUS_INEPRO_regQuantity[PARENT_EO_ID, i];
		regValueType[i]:=MODBUS_INEPRO_regValueType[PARENT_EO_ID, i];

	END_IF

END_FOR
END_ACTION
ACTION Stm:
CASE state OF

	WAIT_STATE:	(* Refresh time manager *)

		ReadTmr(IN:=NOT(ReadTmr.Q));
		IF ReadTmr.Q THEN

			ReadTmr.PT := timing;			(* Refresh timer range *)

			(* Reset state machine variables and counters *)
			retry	:= 0;
			last_state	:= WAIT_STATE;

			(* Start state machine	*)
			state := QUERY_START_CYCLE;

		END_IF

	QUERY_START_CYCLE:
		IF NOT ModBus.MB_Start AND (NOT ModBus.MB_Lock OR retry>0) THEN
			ModBus.MB_Lock := TRUE;

			ModBus.MB_Obj := PARENT_EO_TYPE;
			ModBus.MB_ObjId := PARENT_EO_ID;

			state := QUERY_MEAS_REQ;
		END_IF

	(****			 MEASUREMENTS			  ****)

	QUERY_MEAS_REQ:
		IF NOT ModBus.MB_Start THEN

				IF regAddress[currentReg] <> 0 THEN

					ModBus.MB_Query.SlaveAddress := Address;
					ModBus.MB_Query.FunctionCode := 16#3;
					ModBus.MB_Query.Read_StartAddress :=regAddress[currentReg];
					ModBus.MB_Query.Read_Quantity := regQuantity[currentReg];
					ModBus.MB_Start := TRUE;

					state := QUERY_MEAS_ANSW;

				ELSE

					currentReg:=currentReg+1;

					IF(currentReg<=MODBUS_INEPRO_MAX_REG) THEN

						state := QUERY_MEAS_REQ;

					ELSE

						currentReg:=1;
						fModbusAlr := FALSE;
						retryErr := 0;
						ModBus.MB_Lock := FALSE;
						fTimeout := FALSE;
						state := WAIT_STATE;

					END_IF

				END_IF
		END_IF


	QUERY_MEAS_ANSW:
		IF NOT ModBus.MB_Start THEN
			IF ModBus.MB_MASTER.bInterfaceError<>0 OR ModBus.MB_MASTER.MB_Error<>0 THEN
				last_state := QUERY_MEAS_ANSW;
				state := ERROR_STATE;
			ELSE

				IF (regValueType[currentReg] = VALUE_REAL ) THEN
					regData[currentReg]:=BUILD_REAL_COPY(ModBus.MB_Resp.Data[1],ModBus.MB_Resp.Data[0]);
				END_IF
				IF (regValueType[currentReg] = VALUE_LONG ) THEN
					regDataWord[currentReg,1]:=ModBus.MB_Resp.Data[0];
					regDataWord[currentReg,2]:=ModBus.MB_Resp.Data[1];
				END_IF

				currentReg:=currentReg+1;

				IF(currentReg<=MODBUS_INEPRO_MAX_REG) THEN

					state := QUERY_MEAS_REQ;

				ELSE
					currentReg:=1;
					fModbusAlr := FALSE;
					retryErr := 0;
					ModBus.MB_Lock := FALSE;
					fTimeout := FALSE;
					state := WAIT_STATE;
				END_IF


			END_IF
		END_IF


	ERROR_STATE:	(* Error state *)

		IF retry < 3 THEN
			retry := retry+1;
			state := last_state;

		ELSE
			ModBus.MB_Lock := FALSE;

			(* Verify if slave is dead *)
			IF retryErr < retryErrMaX THEN
				retryErr := retryErr + 1;
			ELSE
				fModbusAlr := TRUE;
			END_IF

			(* Back to wait state *)
			state := WAIT_STATE;

			fTimeout := TRUE;
		END_IF

		IF ModBus.MB_MASTER.MB_Error=MB_TIME_OUT THEN
			state := state;
		END_IF
ELSE
	state := WAIT_STATE;
END_CASE
END_ACTION

(* POU ClevergyBlocks/obj_MODBUS_ANZ, ST *)
FUNCTION_BLOCK obj_MODBUS_ANZ
(* === MODBUS PROTOCOL INTERFACE ===
   v1.1[19/06/15] - Added new VARS allocation and searching
*)
VAR CONSTANT
	VARS_Max	: BYTE := 32;
END_VAR
VAR_INPUT
	(* Settings *)
	ID			: BYTE;
	COM			: BYTE;
	BAUDRATE	: COM_BAUDRATE;
	RS485		: BOOL := FALSE;
	PARITY : COM_PARITY:=PARITY_NO;
	STOP_BITS :COM_STOPBITS:=STOPBITS_2;
	TIME_OUT_TIME : TIME:=t#500ms;

	(* Interface *)
	MB_MASTER	: MODBUS_EXTENDED_MASTER;
	MB_Start	: BOOL;
	MB_Query	: typModbusExtendedQuery;
	MB_Resp		: typModbusResponse;
	MB_Lock		: BOOL;
	MB_Obj		: en_SYS_Objects;
	MB_ObjId	: BYTE;

	(* Variables management *)
	VARS_En		: BOOL := FALSE;
	VARS		: ARRAY [0..VARS_Max] OF typ_MODBUS_VAR_anz;
	VARS_Check	: BOOL;
	VARS_Alarm	: BOOL;

	(* Variables allocation *)
	VAR_Pointer : POINTER TO ARRAY[0..99] OF WORD;
	VAR_Cfg		: POINTER TO typ_MODBUS_VAR_ANZ;
END_VAR
VAR_OUTPUT
	(* Status *)
	Status_Log	: BYTE;
	Status_Vis	: DWORD;
END_VAR
VAR
	sta         : BYTE :=0;
	i			: BYTE;
	j			: BYTE;

	AlarmCOM	: FLT_EVENT;	(* Physical error relative to serial port -> COM	*)
	AlarmMDB	: FLT_EVENT;	(* ModBus error due to communication protocol error	*)

	VarTmr		: TON := (PT:=T#1s);
	VarSta		: BYTE; (* Status *)
	VarCnt		: BYTE; (* Scan counter *)
	VarRetry	: BYTE;
	VarAlarm	: BYTE; (* Last variable with errors *)
END_VAR
MB_MASTER(ENABLE:=TRUE,	ASCII_Mode:=FALSE, bCOM_PORT:=COM, cbCOM_BAUDRATE:=BAUDRATE, cpCOM_PARITY:=PARITY,
		csCOM_STOPBITS:=STOP_BITS,	cbsCOM_BYTESIZE:=BS_8, cfCOM_FLOW_CONTROL:=SEL(RS485,NO_FLOW_CONTROL,HALFDUPLEX),
		tTIME_OUT:=TIME_OUT_TIME,	StartFunction:=MB_Start, ExtQuery:=MB_Query, Response:=MB_Resp);

(* Process variable management *)
IF VARS_En THEN VARS_Process(); END_IF

(* Check status *)
AlarmCOM(IN:=(MB_MASTER.bInterfaceError<>0));
IF AlarmCOM.EVH THEN
	LogEv(SEL(MB_MASTER.bInterfaceError<>3,EL_Wrn,EL_Alarm),EO_MODBUS,ID,1,BYTE_TO_STRING(MB_MASTER.bInterfaceError));
END_IF
IF AlarmCOM.EVL THEN								(* Trigger a fall edge: MODBUS back working *)
	LogEv(EL_Log,EO_MODBUS,ID,2,'MODBUS_OK');
END_IF

(* If VARS not active check if a protocol error has occured (if VARS active this check is already done in "VARS_Process"	*)
IF NOT VARS_En THEN

	AlarmMDB(IN:=(MB_MASTER.MB_Error<>0));
(*	IF AlarmMDB.EVH THEN
		LogEv(EL_Wrn,EO_MODBUS,ID,2,INT_TO_STRING(MB_MASTER.MB_Error));
	END_IF
	IF AlarmMDB.EVL THEN								(* Trigger a fall edge: MODBUS back working *)
		LogEv(EL_Log,EO_MODBUS,ID,2,'MODBUS_OK');
	END_IF
*)
END_IF

(* Log/visu status *)
IF AlarmCOM.IN THEN Status_Log:=2; Status_Vis:=COLOR_RED;
ELSIF Vars_Alarm OR AlarmMDB.IN THEN Status_Log:=1; Status_Vis:=COLOR_YELLOW;
ELSE Status_Log:=0; Status_Vis:=COLOR_GREEN;
END_IF
END_FUNCTION_BLOCK
ACTION VAR_Search:
(* Search VAR with specific pointer if not found return first free VAR
	[Last VAR is not active... used as safe area...] 
*)
j:=VARS_Max;
FOR i := 0 TO VARS_Max-1 DO
	IF VARS[i].Variable=0 AND j>i THEN j:=i; END_IF
	IF VARS[i].Variable=VAR_Pointer THEN
		VAR_Cfg:=ADR(VARS[i]);
		RETURN;
	END_IF
END_FOR
VAR_Cfg:=ADR(VARS[j]);
END_ACTION
ACTION VARS_Process:
(* Update var timers *)
VarTmr(IN:=(NOT VarTmr.Q));
IF VarTmr.Q THEN
	FOR i := 0 TO VARS_Max DO
		IF VARS[i].Refresh_Cnt>0 THEN VARS[i].Refresh_Cnt:=VARS[i].Refresh_Cnt-1; END_IF
	END_FOR
	VARS_Check:=TRUE;
END_IF


(* Process status *)
CASE VarSta OF
	0: (* === Init *)
		VarCnt:=0;
		VarSta:=1;

	1: (* === Wait check signal *)
		IF VARS_Check THEN				(* Decremented "Refresh_Cnt" *)
			VARS_Check:=FALSE;
			VarCnt:=0;
			VarSta:=2;
		END_IF

	2: (* === Check loop *)
		IF NOT (MB_Lock OR MB_Start) THEN
			WHILE VarCnt<=(VARS_Max-1) AND VarSta=2 DO
				(* Check only active vars *)
				IF VARS[VarCnt].Variable<>0 THEN			(* "Variable" is a pointer to word, so if 0 no address *)
					(* Check var auto-refresh on timer checks *)
					IF VARS[VarCnt].Refresh_Time>0 AND VARS[VarCnt].Refresh_Cnt=0 THEN
						VARS[VarCnt].Refresh_Cnt:=VARS[VarCnt].Refresh_Time;
						VarSta:=3;
					END_IF
					(* Check refresh for change or request *)
					CASE VARS[VarCnt].FunCode OF
						5,6,15,16: (* Write functions *)
							IF VARS[VarCnt].Variable_Size=1 THEN
								IF VARS[VarCnt].Variable^[0]<>VARS[VarCnt].Variable_Mirror THEN
									VARS[VarCnt].Variable_Mirror:=VARS[VarCnt].Variable^[0];
									VarSta:=3;
								END_IF
							ELSE
								IF VARS[VarCnt].Variable_Mirror<>0 THEN
									VARS[VarCnt].Variable_Mirror:=0;
									VarSta:=3;
								END_IF
							END_IF
						1,2,3,4: (* Read functions *)
							IF VARS[VarCnt].Variable_Mirror<>0 THEN
								VARS[VarCnt].Variable_Mirror:=0;
								VarSta:=3;
							END_IF
					END_CASE
				END_IF
				(* Process query *)
				IF VarSta=3 THEN
					MB_Lock:=TRUE;
					MB_Query.SlaveAddress:=VARS[VarCnt].SlaveAddress;
					MB_Query.FunctionCode:=VARS[VarCnt].FunCode;
					CASE VARS[VarCnt].FunCode OF
						16#5,16#6,16#F,16#10:
							MB_Query.Read_Quantity:=0;
							MB_Query.Read_StartAddress:=0;
							MB_Query.Write_StartAddress:=VARS[VarCnt].FunAddress;
							MB_Query.Write_Quantity:=VARS[VarCnt].Variable_Size;
							IF VARS[VarCnt].Variable_Size=200 THEN
								COPY_32SWAP16(VARS[VarCnt].Variable, ADR(MB_Query.Write_Data[0]));
							ELSIF VARS[VarCnt].Variable_Size>1 THEN
								MEMCPY(VARS[VarCnt].Variable, ADR(MB_Query.Write_Data[0]), 2*VARS[VarCnt].Variable_Size);
							ELSE
								MB_Query.Write_Data[0]:=VARS[VarCnt].Variable^[0];
							END_IF
						16#1,16#2,16#3,16#4:
							MB_Query.Read_StartAddress:=VARS[VarCnt].FunAddress;
							IF VARS[VarCnt].Variable_Size=200 THEN MB_Query.Read_Quantity:=2; ELSE
							  MB_Query.Read_Quantity:=VARS[VarCnt].Variable_Size;
							END_IF
							MB_Query.Write_StartAddress:=0;
							MB_Query.Write_Quantity:=0;
					END_CASE
					VarRetry:=0;
					MB_Start:=TRUE;
				ELSE
					VarCnt:=VarCnt+1;
				END_IF
			END_WHILE
			(* Check loop completed -> no actions *)
			IF VarSta=2 THEN VarSta:=1; END_IF
		END_IF

	3: (* === Wait & process MB response *)
		IF NOT MB_Start THEN
			IF MB_MASTER.MB_Error=0 THEN
				CASE VARS[VarCnt].FunCode OF
					1,2,3,4:
						IF VARS[VarCnt].Variable_Size=200 THEN
							COPY_32SWAP16(ADR(MB_Resp.Data), VARS[VarCnt].Variable);
						ELSIF VARS[VarCnt].Variable_Size>1 THEN
							MEMCPY(ADR(MB_Resp.Data), VARS[VarCnt].Variable, 2*VARS[VarCnt].Variable_Size);
						ELSE
							VARS[VarCnt].Variable^[0]:=MB_Resp.Data[0];
						END_IF
				END_CASE
				MB_Lock:=FALSE;
				(* Signal error recovery *)
				IF VARS_Alarm=TRUE AND VarCnt=VarAlarm THEN
					LogEv(EL_Wrn,EO_MODBUS,ID,5,'');
					VARS_Alarm:=FALSE;
				END_IF
				(* Next var *)
				VarCnt:=VarCnt+1;
				VarSta:=2;
			ELSE
				IF VarRetry<3 THEN
					VarRetry:=VarRetry+1;
					MB_Start:=TRUE;
				ELSE
					MB_Lock:=FALSE;
					(* Signal error *)
					IF VARS_Alarm=FALSE THEN
						LogEv(EL_Wrn,EO_MODBUS,ID,3,INT_TO_STRING(MB_MASTER.MB_Error));
						VARS_Alarm:=TRUE;
						VarAlarm:=VarCnt-1;
					END_IF
					(* Next var *)
					VarCnt:=VarCnt+1;
					VarSta:=2;
				END_IF
			END_IF
		END_IF

ELSE
	VarSta:=0;
END_CASE
END_ACTION

(* POU Plant_Objects/obj_COMPRESSORE_NEW, ST *)
FUNCTION_BLOCK obj_COMPRESSORE_NEW
VAR CONSTANT

	TimeOutModBus: TON;


END_VAR
VAR_INPUT
	ID			:	BYTE;
	Address		:	BYTE;


	(* Modbus *)
	Refresh_Now	:	BOOL;			(* Richiesta di lettura stato macchina Immediata  *)
	retryErrMax	:	BYTE := 2;

	OnOff		: 	BOOL;

	IndirizzoDaScrivere: WORD;
	DatoDaScrivere: INT;
	ScriviDato: BOOL;
	ScriviCoil: BOOL;

	fWriteAttivazioneComandi:BOOL;

	RUN_REQ: BOOL;
	STOP_REQ:BOOL;
	AgggiornoStartStop: BOOL;
	CARICO_REQ: BOOL;
	RELEASE_REQ: BOOL;
END_VAR
VAR_IN_OUT
	ModBus		:obj_MODBUS;
END_VAR
VAR_OUTPUT
	Run			:	BOOL;

	Status_Log	:	WORD;
	Status_Vis	:	DWORD;
END_VAR
VAR
	(* da diego per gestione stato stringa > 255*)
	temp :STRING(255);
	tempRaw		: ARRAY [0..MAX_SEND_TCP_CLIENT] OF BYTE;
	tempRawLen :DINT;
	longString:STRING(255);

	(* Timer manage switch on/off delay *)
	Delay		: 	TONOF;
	Warning		:	FLT_TAP := (TAP:=100);
	AllarmeCompressore_MB		:	FLT_TAP;
	WarningCompressore_MB		:	FLT_TAP;

	state		:	INT;
	retry		:	BYTE;
	retryErr	:	BYTE;
	ReadTmr		:	TON := (PT:=T#5s);
	fModbusAlr:BOOL;

	Ctrl_Run: BOOL;


	VerificaFuctionCode: INT;
	VerificaNodoLetto: INT;
	ErroreComuModBus: BOOL;
	IndiceErrore: BYTE;

	MB_BitStato: ARRAY [0..1] OF BOOL;
	MB_RegistriLetti: ARRAY [0..1] OF INT;
	MB_RegistriHoldingLetti: ARRAY [0..260] OF INT;
	MB_BitStatoCoil: ARRAY [0..1] OF BOOL;



	AddressRead: BYTE;
	index: BYTE;
	indexErr: BYTE;





	x: INT;
	moreno1: INT;
	moreno2: INT;
	IndirizzoStart: INT;
	Stop: BOOL;
	start: BOOL;
	StatusControl: ARRAY [0..15] OF BOOL;
END_VAR
(* Call ModBus state machine *)
Stm();

(* Check alarm	*)
CheckAlarm();

(* Seganalzione stato Compressore  *)
IF ErroreComuModBus THEN
		Status_Log:=2; Status_Vis:=16#2020F0;
  ELSIF WarningCompressore_MB.IN  THEN
		Status_Log:=1; Status_Vis:=16#20F0F0;
    ELSE
		Status_Log:=0;
		Status_Vis:=16#006000;
END_IF
END_FUNCTION_BLOCK
ACTION AddLogData:
Logger.s1:=INSERT('&COMPINGRR=',BYTE_TO_STRING(ID),10);
IF ID<10 THEN Logger.s1:=INSERT(Logger.s1,'0',10); END_IF

FOR tempRawLen:=0 TO MAX_SEND_TCP_CLIENT DO
                tempRaw[tempRawLen]:=0;
END_FOR

tempRawLen:=0;


temp:=Logger.s1;
ADDSTRING(ADR(tempRaw), ADR(temp), tempRawLen);

temp:=CONCAT(WORD_TO_STRING(Status_Log),';');
ADDSTRING(ADR(tempRaw), ADR(temp), tempRawLen);


(* Sparo gli ingressi Digitali **)
FOR x:= 0 TO 15 DO
	temp:=CONCAT(SEL(StatusControl[x],'0','1'),';');
	ADDSTRING(ADR(tempRaw), ADR(temp), tempRawLen);
END_FOR

(*

temp:=CONCAT(INT_TO_STRING(MB_RegistriHoldingLetti[1]),';');
ADDSTRING(ADR(tempRaw), ADR(temp), tempRawLen); *)
temp:=CONCAT(INT_TO_STRING(MB_RegistriHoldingLetti[3]),';');
ADDSTRING(ADR(tempRaw), ADR(temp), tempRawLen);
temp:=CONCAT(INT_TO_STRING(MB_RegistriHoldingLetti[4]),';');
ADDSTRING(ADR(tempRaw), ADR(temp), tempRawLen);
temp:=CONCAT(INT_TO_STRING(MB_RegistriHoldingLetti[5]),';');
ADDSTRING(ADR(tempRaw), ADR(temp), tempRawLen);
temp:=CONCAT(INT_TO_STRING(MB_RegistriHoldingLetti[6]),';');
ADDSTRING(ADR(tempRaw), ADR(temp), tempRawLen);
temp:=CONCAT(INT_TO_STRING(MB_RegistriHoldingLetti[11]),';');
ADDSTRING(ADR(tempRaw), ADR(temp), tempRawLen);
temp:=CONCAT(INT_TO_STRING(MB_RegistriHoldingLetti[12]),';');
ADDSTRING(ADR(tempRaw), ADR(temp), tempRawLen);
temp:=CONCAT(INT_TO_STRING(MB_RegistriHoldingLetti[13]),';');
ADDSTRING(ADR(tempRaw), ADR(temp), tempRawLen);
temp:=CONCAT(INT_TO_STRING(MB_RegistriHoldingLetti[14]),';');
ADDSTRING(ADR(tempRaw), ADR(temp), tempRawLen);
temp:=CONCAT(INT_TO_STRING(MB_RegistriHoldingLetti[15]),';');
ADDSTRING(ADR(tempRaw), ADR(temp), tempRawLen);
temp:=CONCAT(INT_TO_STRING(MB_RegistriHoldingLetti[19]),';');
ADDSTRING(ADR(tempRaw), ADR(temp), tempRawLen);
temp:=CONCAT(INT_TO_STRING(MB_RegistriHoldingLetti[20]),';');
ADDSTRING(ADR(tempRaw), ADR(temp), tempRawLen);
temp:=CONCAT(INT_TO_STRING(MB_RegistriHoldingLetti[25]),';');
ADDSTRING(ADR(tempRaw), ADR(temp), tempRawLen);
temp:=CONCAT(INT_TO_STRING(MB_RegistriHoldingLetti[26]),';');
ADDSTRING(ADR(tempRaw), ADR(temp), tempRawLen);
temp:=CONCAT(INT_TO_STRING(MB_RegistriHoldingLetti[27]),';');
ADDSTRING(ADR(tempRaw), ADR(temp), tempRawLen);
temp:=CONCAT(INT_TO_STRING(MB_RegistriHoldingLetti[30]),';');
ADDSTRING(ADR(tempRaw), ADR(temp), tempRawLen);
temp:=CONCAT(INT_TO_STRING(MB_RegistriHoldingLetti[31]),';');
ADDSTRING(ADR(tempRaw), ADR(temp), tempRawLen);
temp:=CONCAT(INT_TO_STRING(MB_RegistriHoldingLetti[64]),';');
ADDSTRING(ADR(tempRaw), ADR(temp), tempRawLen);
temp:=CONCAT(INT_TO_STRING(MB_RegistriHoldingLetti[65]),';');
ADDSTRING(ADR(tempRaw), ADR(temp), tempRawLen);
temp:=CONCAT(INT_TO_STRING(MB_RegistriHoldingLetti[101]),';');
ADDSTRING(ADR(tempRaw), ADR(temp), tempRawLen);
temp:=CONCAT(INT_TO_STRING(MB_RegistriHoldingLetti[112]),';');
ADDSTRING(ADR(tempRaw), ADR(temp), tempRawLen);
temp:=CONCAT(INT_TO_STRING(MB_RegistriHoldingLetti[113]),';');
ADDSTRING(ADR(tempRaw), ADR(temp), tempRawLen);
temp:=CONCAT(INT_TO_STRING(MB_RegistriHoldingLetti[114]),';');
ADDSTRING(ADR(tempRaw), ADR(temp), tempRawLen);
temp:=CONCAT(INT_TO_STRING(MB_RegistriHoldingLetti[115]),';');
ADDSTRING(ADR(tempRaw), ADR(temp), tempRawLen);
temp:=CONCAT(INT_TO_STRING(MB_RegistriHoldingLetti[118]),';');
ADDSTRING(ADR(tempRaw), ADR(temp), tempRawLen);
temp:=CONCAT(INT_TO_STRING(MB_RegistriHoldingLetti[119]),';');
ADDSTRING(ADR(tempRaw), ADR(temp), tempRawLen);
temp:=CONCAT(INT_TO_STRING(MB_RegistriHoldingLetti[121]),';');
ADDSTRING(ADR(tempRaw), ADR(temp), tempRawLen);
temp:=CONCAT(INT_TO_STRING(MB_RegistriHoldingLetti[255]),';');
ADDSTRING(ADR(tempRaw), ADR(temp), tempRawLen);
temp:=(INT_TO_STRING(MB_RegistriHoldingLetti[256]));
ADDSTRING(ADR(tempRaw), ADR(temp), tempRawLen);


ADDSTRING(ADR(Logger.TData), ADR(tempRaw), Logger.TLen);
END_ACTION
ACTION CheckAlarm:
(**** GEstione Log ad Evento *****)




	AllarmeCompressore_MB(IN:=MB_RegistriHoldingLetti[1].6 );

	IF AllarmeCompressore_MB.EVH THEN
		LogEv(EL_Alarm,EO_COMPINGRR,ID,1,CONCAT ('AllarmeAttivo_n.', INT_TO_STRING(MB_RegistriHoldingLetti[255])));
	END_IF

	IF AllarmeCompressore_MB.EVL THEN
		LogEv(EL_Log,EO_COMPINGRR,ID,2,CONCAT ('AllarmeRientrato_n.', INT_TO_STRING(MB_RegistriHoldingLetti[255])));
	END_IF



	WarningCompressore_MB(IN:=MB_RegistriHoldingLetti[1].5 );

	IF WarningCompressore_MB.EVH THEN
		LogEv(EL_Wrn,EO_COMPINGRR,ID,1,CONCAT ('AllarmeAttivo_n.', INT_TO_STRING(MB_RegistriHoldingLetti[255])));
	END_IF

	IF WarningCompressore_MB.EVL THEN
		LogEv(EL_Log,EO_COMPINGRR,ID,2,CONCAT ('AllarmeRientrato_n.', INT_TO_STRING(MB_RegistriHoldingLetti[255])));
	END_IF
END_ACTION
ACTION Stm:
CASE state OF
	0:	(* Refresh time manager *)
		ReadTmr(IN:=NOT ReadTmr.Q);
		(*A tempo interrogo il nodo sempre che non ci sia qualcuno che lo sta interrogando in quel momento *)

		IF (ReadTmr.Q AND NodoDaInterrogareCompressoreNuovo=Address )  AND NOT InibiscoModbusCompressoreNuovo THEN
			state := 10;
			ReadTmr.PT := T#100ms;  (* moreno *)
			Refresh_Now := FALSE;
			InibiscoModbusCompressoreNuovo := TRUE;
		END_IF

	(**** Leggo le Analogiche a Disposzione  ****)

	10:	(* richiedo lettura Holding Registere   *)

		Modbus.MB_Query.SlaveAddress := Address;
		Modbus.MB_Query.FunctionCode := 3;
		IndirizzoStart:=1;
		ModBus.MB_Query.Read_StartAddress :=IndirizzoStart - 1 ;
		ModBus.MB_Query.Read_Quantity := 19;(*19;*)
		ModBus.MB_Start := TRUE;
		state := 20;

	20:	(* Risposta all'interrogazione *)
		IF NOT ModBus.MB_Start   THEN
			VerificaFuctionCode:=ModBus.MB_Resp.FunctionCode;
			VerificaNodoLetto:=ModBus.MB_Resp.SlaveAddress;

			IF ModBus.MB_MASTER.MB_Error<>0 THEN
				state := 300;
			ELSE
				FOR x:=0 TO ModBus.MB_Query.Read_Quantity DO
					MB_RegistriHoldingLetti[x+IndirizzoStart] := ModBus.MB_Resp.Data[x];   	(* Vedi tabella *)
				END_FOR

				(* trasforo la wordo in singoli 16 bit *)

					StatusControl[0]:= MB_RegistriHoldingLetti[IndirizzoStart].0;   	(* Vedi tabella *)
					StatusControl[1]:= MB_RegistriHoldingLetti[IndirizzoStart].1;   	(* Vedi tabella *)
					StatusControl[2]:= MB_RegistriHoldingLetti[IndirizzoStart].2;   	(* Vedi tabella *)
					StatusControl[3]:= MB_RegistriHoldingLetti[IndirizzoStart].3;   	(* Vedi tabella *)
					StatusControl[4]:= MB_RegistriHoldingLetti[IndirizzoStart].4;   	(* Vedi tabella *)
					StatusControl[5]:= MB_RegistriHoldingLetti[IndirizzoStart].5;   	(* Vedi tabella *)
					StatusControl[6]:= MB_RegistriHoldingLetti[IndirizzoStart].6;   	(* Vedi tabella *)
					StatusControl[7]:= MB_RegistriHoldingLetti[IndirizzoStart].7;   	(* Vedi tabella *)
					StatusControl[8]:= MB_RegistriHoldingLetti[IndirizzoStart].8;   	(* Vedi tabella *)
					StatusControl[9]:= MB_RegistriHoldingLetti[IndirizzoStart].9;   	(* Vedi tabella *)
					StatusControl[10]:= MB_RegistriHoldingLetti[IndirizzoStart].10;   	(* Vedi tabella *)
					StatusControl[11]:= MB_RegistriHoldingLetti[IndirizzoStart].11;   	(* Vedi tabella *)
					StatusControl[12]:= MB_RegistriHoldingLetti[IndirizzoStart].12;   	(* Vedi tabella *)
					StatusControl[13]:= MB_RegistriHoldingLetti[IndirizzoStart].13;   	(* Vedi tabella *)
					StatusControl[14]:= MB_RegistriHoldingLetti[IndirizzoStart].14;   	(* Vedi tabella *)
					StatusControl[15]:= MB_RegistriHoldingLetti[IndirizzoStart].15;   	(* Vedi tabella *)





				IndirizzoStart:=20;
				ModBus.MB_Query.Read_StartAddress :=IndirizzoStart - 1 ;
				ModBus.MB_Query.Read_Quantity := 19;
				ModBus.MB_Start := TRUE;

				state := 30;
			END_IF
		END_IF

	30: (* Rispota Altri paramenti *)
		IF NOT ModBus.MB_Start  THEN

			IF ModBus.MB_MASTER.MB_Error<>0 THEN
				state := 300;
			ELSE

				FOR x:=0 TO ModBus.MB_Query.Read_Quantity DO
					MB_RegistriHoldingLetti[x+IndirizzoStart] := ModBus.MB_Resp.Data[x];   	(* Vedi tabella *)
				END_FOR

				IndirizzoStart:=40;
				ModBus.MB_Query.Read_StartAddress :=IndirizzoStart - 1 ;
				ModBus.MB_Query.Read_Quantity := 19;
				ModBus.MB_Start := TRUE;

				state := 35;
			END_IF
		END_IF
	35: (* Rispota Altri paramenti *)
		IF NOT ModBus.MB_Start  THEN

			IF ModBus.MB_MASTER.MB_Error<>0 THEN
				state := 300;
			ELSE

				FOR x:=0 TO ModBus.MB_Query.Read_Quantity DO
					MB_RegistriHoldingLetti[x+IndirizzoStart] := ModBus.MB_Resp.Data[x];   	(* Vedi tabella *)
				END_FOR

				IndirizzoStart:=64;
				ModBus.MB_Query.Read_StartAddress :=IndirizzoStart - 1 ;
				ModBus.MB_Query.Read_Quantity := 6;
				ModBus.MB_Start := TRUE;

				state := 40;
			END_IF
		END_IF
	40: (* Rispota Altri paramenti *)
		IF NOT ModBus.MB_Start  THEN

			IF ModBus.MB_MASTER.MB_Error<>0 THEN
				state := 300;
			ELSE

				FOR x:=0 TO ModBus.MB_Query.Read_Quantity DO
					MB_RegistriHoldingLetti[x+IndirizzoStart] := ModBus.MB_Resp.Data[x];   	(* Vedi tabella *)
				END_FOR

				IndirizzoStart:=90;
				ModBus.MB_Query.Read_StartAddress :=IndirizzoStart - 1 ;
				ModBus.MB_Start := TRUE;

				state := 45;
			END_IF
		END_IF

	45: (* Rispota Altri paramenti *)
		IF NOT ModBus.MB_Start  THEN

			IF ModBus.MB_MASTER.MB_Error<>0 THEN
				state := 300;
			ELSE
				FOR x:=0 TO ModBus.MB_Query.Read_Quantity DO
					MB_RegistriHoldingLetti[x+IndirizzoStart] := ModBus.MB_Resp.Data[x];   	(* Vedi tabella *)
				END_FOR

				IndirizzoStart:=110;
				ModBus.MB_Query.Read_StartAddress :=IndirizzoStart - 1 ;
				ModBus.MB_Query.Read_Quantity := 19;
				ModBus.MB_Start := TRUE;

				state := 50;
			END_IF
		END_IF


	50: (* Rispota Altri paramenti *)
		IF NOT ModBus.MB_Start  THEN

			IF ModBus.MB_MASTER.MB_Error<>0 THEN
				state := 300;
			ELSE
				FOR x:=0 TO ModBus.MB_Query.Read_Quantity DO
					MB_RegistriHoldingLetti[x+IndirizzoStart] := ModBus.MB_Resp.Data[x];   	(* Vedi tabella *)
				END_FOR

				IndirizzoStart:=130;
				ModBus.MB_Query.Read_StartAddress :=IndirizzoStart - 1 ;
				ModBus.MB_Query.Read_Quantity := 5;
				ModBus.MB_Start := TRUE;


				state := 55;
			END_IF
		END_IF

	55: (* Rispota Altri paramenti *)
		IF NOT ModBus.MB_Start  THEN

			IF ModBus.MB_MASTER.MB_Error<>0 THEN
				state := 300;
			ELSE
				FOR x:=0 TO ModBus.MB_Query.Read_Quantity DO
					MB_RegistriHoldingLetti[x+IndirizzoStart] := ModBus.MB_Resp.Data[x];   	(* Vedi tabella *)
				END_FOR

				IndirizzoStart:=240;
				ModBus.MB_Query.Read_StartAddress :=IndirizzoStart - 1 ;
				ModBus.MB_Query.Read_Quantity := 3;
				ModBus.MB_Start := TRUE;

				state := 60;
			END_IF
		END_IF

	60: (* Rispota Altri paramenti *)
		IF NOT ModBus.MB_Start  THEN

			IF ModBus.MB_MASTER.MB_Error<>0 THEN
				state := 300;
			ELSE
				FOR x:=0 TO ModBus.MB_Query.Read_Quantity DO
					MB_RegistriHoldingLetti[x+IndirizzoStart] := ModBus.MB_Resp.Data[x];   	(* Vedi tabella *)
				END_FOR

				state :=290;
			END_IF
		END_IF


		290:    (* Scrittura il comando di run o stop da remoto*)
		IF NOT ModBus.MB_Start THEN
			IF ModBus.MB_MASTER.MB_Error<>0 THEN (*OR ModBus.MB_MASTER.MB_Error<>0 THEN*)
				state := 300;
			ELSE
				IF AgggiornoStartStop  THEN

					Modbus.MB_Query.FunctionCode := 6;
					Modbus.MB_Query.SlaveAddress := Address;
					ModBus.MB_Query.Write_Quantity :=1;


					IF RUN_REQ THEN
							IndirizzoDaScrivere:=1;
							 DatoDaScrivere:=MB_RegistriHoldingLetti[IndirizzoDaScrivere];
	  							 DatoDaScrivere.0:=TRUE;
  							        DatoDaScrivere.1:=TRUE;
							        DatoDaScrivere.2:=TRUE;
								 RUN_REQ:=FALSE;
					END_IF
					IF STOP_REQ THEN
							IndirizzoDaScrivere:=1;
								 DatoDaScrivere:=MB_RegistriHoldingLetti[IndirizzoDaScrivere];
	  							 DatoDaScrivere.0:=TRUE;
  							        DatoDaScrivere.1:=FALSE;
							        DatoDaScrivere.2:=TRUE;
								 STOP_REQ:=FALSE;
					END_IF
					IF RELEASE_REQ THEN
							IndirizzoDaScrivere:=1;
								 DatoDaScrivere:=MB_RegistriHoldingLetti[IndirizzoDaScrivere];
	  							 DatoDaScrivere.0:=FALSE;
  							        DatoDaScrivere.1:=FALSE;
							        DatoDaScrivere.2:=TRUE;
								 RELEASE_REQ:=FALSE;
					END_IF
			(*		IF CARICO_REQ THEN
								IndirizzoDaScrivere:=1;
							 DatoDaScrivere:=MB_RegistriHoldingLetti[IndirizzoDaScrivere];
	  							 DatoDaScrivere.0:=TRUE;
  							        DatoDaScrivere.1:=TRUE;
							        DatoDaScrivere.2:= NOT DatoDaScrivere.2;
								 CARICO_REQ:=FALSE;
					END_IF  *)

					ModBus.MB_Query.Write_StartAddress := IndirizzoDaScrivere-1;
					ModBus.MB_Query.Write_Data[0] := DatoDaScrivere;
					ModBus.MB_Start := TRUE;
					state := 295;
					AgggiornoStartStop:=FALSE;
				ELSE
					state := 295;
				END_IF
			END_IF
		END_IF
(*		291:    (* Scrittura BOOL - COIL o WORD *)
		IF NOT ModBus.MB_Start THEN
			IF ModBus.MB_MASTER.MB_Error<>0 THEN (*OR ModBus.MB_MASTER.MB_Error<>0 THEN*)
				state := 300;
			ELSE
				IF ScriviDato THEN
					IF ScriviCoil THEN
						Modbus.MB_Query.FunctionCode := 5;
					ELSE
						Modbus.MB_Query.FunctionCode := 6;
					END_IF
					Modbus.MB_Query.SlaveAddress := Address;
					ModBus.MB_Query.Write_StartAddress := IndirizzoDaScrivere-1;
					ModBus.MB_Query.Write_Quantity :=1;
					ModBus.MB_Query.Write_Data[0] := DatoDaScrivere;
					ModBus.MB_Start := TRUE;
						IF ScriviCoil THEN
							IF 	MB_BitStato[IndirizzoDaScrivere]=WORD_TO_BOOL(DatoDaScrivere-1) THEN
								ScriviDato:=FALSE;
							END_IF
						ELSE
							IF 	MB_RegistriHoldingLetti[IndirizzoDaScrivere]=DatoDaScrivere THEN
								ScriviDato:=FALSE;
							END_IF
						END_IF
					state := 295;
				ELSE
					state := 295;
				END_IF
			END_IF
		END_IF

*)


		295:
		IF NOT ModBus.MB_Start THEN
			IF ModBus.MB_MASTER.MB_Error<>0 THEN (*OR ModBus.MB_MASTER.MB_Error<>0 THEN*)
				state := 300;
			ELSE
				IF fModbusAlr THEN fModbusAlr := FALSE; END_IF
				NodoDaInterrogareCompressoreNuovo:=Address+1;
				InibiscoModbusCompressoreNuovo:=FALSE;
				retryErr := 0;
				retry := 0;
				state := 0;
					IF fModbusAlr=FALSE AND ErroreComuModBus=TRUE THEN
						LogEv(EL_Log,EO_COMPINGRML,ID,62,'ComunicazioneModBus_OK');
						ErroreComuModBus := FALSE;
				(*	WarningCtr := SEL(WarningCtr=0, WarningCtr-1, 0); *)
					END_IF
			END_IF


		END_IF




	(**** CHECK MODBUS ERROR ****)
	300: 	(* Release MODBUS *)
			InibiscoModbusCompressoreNuovo:=FALSE;
			(* Retries *)
			retry:=retry+1;
			IF retry>3 THEN
				retry:=0;

				(* Verify if slave is dead *)
				IF retryErr < retryErrMaX THEN
					retryErr := retryErr + 1;
				ELSE
					fModbusAlr := TRUE;
					(* Verify ModBus error	*)

					IF fModbusAlr AND ErroreComuModBus=FALSE THEN
						LogEv(EL_Alarm,EO_COMPINGRML,ID,61,CONCAT('ErroreModbus_',INT_TO_STRING(ModBus.MB_MASTER.MB_Error)));
						ErroreComuModBus := TRUE;
					END_IF
				END_IF

				END_IF
			Refresh_Now := FALSE;
			NodoDaInterrogareCompressoreNuovo:=Address+1;
			state:=0;
END_CASE




(* Controllo Time Out Ciclo ModBus *)

TimeOutModBus(In:=state<>0,PT:=t#3s);
IF TimeOutModBus.Q THEN
	State:=0;
	Refresh_Now:=TRUE;  (* Rilancio la lettura del nodo *)
	IF MODBUS.MB_Lock=TRUE THEN MODBUS.MB_Lock:=FALSE;END_IF
	IF InibiscoModbusCompressoreNuovo=TRUE THEN InibiscoModbusCompressoreNuovo:=FALSE;END_IF
	NodoDaInterrogareCompressoreNuovo:=Address+1;

END_IF
END_ACTION

(* POU Plant_Objects/obj_MODBUS, ST *)
FUNCTION_BLOCK obj_MODBUS
(* === MODBUS PROTOCOL INTERFACE ===
   v1.1[19/06/15] - Added new VARS allocation and searching
*)
VAR CONSTANT
	VARS_Max	: BYTE := 32;
END_VAR
VAR_INPUT
	(* Settings *)
	ID			: BYTE;
	COM			: BYTE;
	BAUDRATE	: COM_BAUDRATE;
	RS485		: BOOL := FALSE;

	N_STOPBits	:BYTE:=1;

 	(* Interface *)
	MB_MASTER	: MODBUS_EXTENDED_MASTER;
	MB_Start	: BOOL;
	MB_Query	: typModbusExtendedQuery;
	MB_Resp		: typModbusResponse;
	MB_Lock		: BOOL;
	MB_timeOut	: TIME := t#500ms;

	(* Variables management *)
	VARS_En		: BOOL;
	VARS		: ARRAY [0..VARS_Max] OF typ_MODBUS_VAR;
	VARS_Check	: BOOL;
	VARS_Alarm	: BOOL;

	(* Variables allocation *)
	VAR_Pointer : POINTER TO ARRAY[0..99] OF WORD;
	VAR_Cfg		: POINTER TO typ_MODBUS_VAR;
END_VAR
VAR_OUTPUT
	(* Status *)
	Status_Log	: BYTE;
	Status_Vis	: DWORD;
END_VAR
VAR
	sta         : BYTE :=0;
	i			: BYTE;
	j			: BYTE;
	Alarm		: FLT_EVENT;
	
	VarTmr		: TON := (PT:=T#1s);
	VarSta		: BYTE; (* Status *)
	VarCnt		: BYTE; (* Scan counter *)
	VarRetry	: BYTE;
	VarAlarm	: BYTE; (* Last variable with errors *)
END_VAR
IF N_STOPBits=1 THEN MB_MASTER.csCOM_STOPBITS:=STOPBITS_1;END_IF
IF N_STOPBits=2 THEN MB_MASTER.csCOM_STOPBITS:=STOPBITS_2;END_IF

MB_MASTER(ENABLE:=TRUE,	ASCII_Mode:=FALSE, bCOM_PORT:=COM, cbCOM_BAUDRATE:=BAUDRATE, cpCOM_PARITY:=PARITY_NO,
		cbsCOM_BYTESIZE:=BS_8, cfCOM_FLOW_CONTROL:=SEL(RS485,NO_FLOW_CONTROL,HALFDUPLEX),
		tTIME_OUT:=MB_timeOut,	StartFunction:=MB_Start, ExtQuery:=MB_Query, Response:=MB_Resp);

(* Process variable management *)
IF VARS_En THEN VARS_Process(); END_IF

(* Check status *)
Alarm(IN:=(MB_MASTER.bInterfaceError<>0));
IF Alarm.EVH THEN
	LogEv(SEL(MB_MASTER.bInterfaceError<>3,EL_Wrn,EL_Alarm),EO_MODBUS,ID,1,BYTE_TO_STRING(MB_MASTER.bInterfaceError));
END_IF
IF Alarm.EVL THEN								(* Trigger a fall edge: MODBUS back working *)
	LogEv(EL_Log,EO_MODBUS,ID,2,'MODBUS_OK');
END_IF

(* Log/visu status *)
   IF Alarm.IN   THEN Status_Log:=2; Status_Vis:=COLOR_RED;
ELSIF Vars_Alarm THEN Status_Log:=1; Status_Vis:=COLOR_YELLOW;
  				 ELSE Status_Log:=0; Status_Vis:=COLOR_GREEN;
END_IF
END_FUNCTION_BLOCK
ACTION VAR_Search:
(* Search VAR with specific pointer if not found return first free VAR
	[Last VAR is not active... used as safe area...] 
*)
j:=VARS_Max;
FOR i := 0 TO VARS_Max-1 DO
	IF VARS[i].Variable=0 AND j>i THEN j:=i; END_IF
	IF VARS[i].Variable=VAR_Pointer THEN
		VAR_Cfg:=ADR(VARS[i]);
		RETURN;
	END_IF
END_FOR
VAR_Cfg:=ADR(VARS[j]);
END_ACTION
ACTION VARS_Process:
(* Update var timers *)
VarTmr(IN:=(NOT VarTmr.Q));
IF VarTmr.Q THEN
	FOR i := 0 TO VARS_Max DO
		IF VARS[i].Refresh_Cnt>0 THEN VARS[i].Refresh_Cnt:=VARS[i].Refresh_Cnt-1; END_IF
	END_FOR
	VARS_Check:=TRUE;
END_IF


(* Process status *)
CASE VarSta OF
	0: (* === Init *)
		VarCnt:=0;
		VarSta:=1;

	1: (* === Wait check signal *)
		IF VARS_Check THEN				(* Decremented "Refresh_Cnt" *)
			VARS_Check:=FALSE;
			VarCnt:=0;
			VarSta:=2;
		END_IF

	2: (* === Check loop *)
		IF NOT (MB_Lock OR MB_Start) THEN
			WHILE VarCnt<=(VARS_Max-1) AND VarSta=2 DO
				(* Check only active vars *)
				IF VARS[VarCnt].Variable<>0 THEN			(* "Variable" is a pointer to word, so if 0 no address *)
					(* Check var auto-refresh on timer checks *)
					IF VARS[VarCnt].Refresh_Time>0 AND VARS[VarCnt].Refresh_Cnt=0 THEN
						VARS[VarCnt].Refresh_Cnt:=VARS[VarCnt].Refresh_Time;
						VarSta:=3;
					END_IF
					(* Check refresh for change or request *)
					CASE VARS[VarCnt].FunCode OF
						5,6,15,16: (* Write functions *)
							IF VARS[VarCnt].Variable_Size=1 THEN
								IF VARS[VarCnt].Variable^<>VARS[VarCnt].Variable_Mirror THEN
									VARS[VarCnt].Variable_Mirror:=VARS[VarCnt].Variable^;
									VarSta:=3;
								END_IF
							ELSE
								IF VARS[VarCnt].Variable_Mirror<>0 THEN
									VARS[VarCnt].Variable_Mirror:=0;
									VarSta:=3;
								END_IF
							END_IF
						1,2,3,4: (* Read functions *)
							IF VARS[VarCnt].Variable_Mirror<>0 THEN
								VARS[VarCnt].Variable_Mirror:=0;
								VarSta:=3;
							END_IF
					END_CASE
				END_IF
				(* Process query *)
				IF VarSta=3 THEN
					MB_Lock:=TRUE;
					MB_Query.SlaveAddress:=VARS[VarCnt].SlaveAddress;
					MB_Query.FunctionCode:=VARS[VarCnt].FunCode;
					CASE VARS[VarCnt].FunCode OF
						16#5,16#6,16#F,16#10:
							MB_Query.Read_Quantity:=0;
							MB_Query.Read_StartAddress:=0;
							MB_Query.Write_StartAddress:=VARS[VarCnt].FunAddress;
							MB_Query.Write_Quantity:=VARS[VarCnt].Variable_Size;
							IF VARS[VarCnt].Variable_Size=200 THEN
								COPY_32SWAP16(VARS[VarCnt].Variable, ADR(MB_Query.Write_Data[0]));
							ELSIF VARS[VarCnt].Variable_Size>1 THEN
								MEMCPY(VARS[VarCnt].Variable, ADR(MB_Query.Write_Data[0]), 2*VARS[VarCnt].Variable_Size);
							ELSE
								MB_Query.Write_Data[0]:=VARS[VarCnt].Variable^;
							END_IF
						16#1,16#2,16#3,16#4:
							MB_Query.Read_StartAddress:=VARS[VarCnt].FunAddress;
							IF VARS[VarCnt].Variable_Size=200 THEN MB_Query.Read_Quantity:=2; ELSE
							  MB_Query.Read_Quantity:=VARS[VarCnt].Variable_Size;
							END_IF
							MB_Query.Write_StartAddress:=0;
							MB_Query.Write_Quantity:=0;
					END_CASE
					VarRetry:=0;
					MB_Start:=TRUE;
				ELSE
					VarCnt:=VarCnt+1;
				END_IF
			END_WHILE
			(* Check loop completed -> no actions *)
			IF VarSta=2 THEN VarSta:=1; END_IF
		END_IF

	3: (* === Wait & process MB response *)
		IF NOT MB_Start THEN
			IF MB_MASTER.MB_Error=0 THEN
				CASE VARS[VarCnt].FunCode OF
					1,2,3,4:
						IF VARS[VarCnt].Variable_Size=200 THEN
							COPY_32SWAP16(ADR(MB_Resp.Data), VARS[VarCnt].Variable);
						ELSIF VARS[VarCnt].Variable_Size>1 THEN
							MEMCPY(ADR(MB_Resp.Data), VARS[VarCnt].Variable, 2*VARS[VarCnt].Variable_Size);
						ELSE
							VARS[VarCnt].Variable^:=MB_Resp.Data[0];
						END_IF
				END_CASE
				MB_Lock:=FALSE;
				(* Signal error recovery *)
				IF VARS_Alarm=TRUE AND VarCnt=VarAlarm THEN
					LogEv(EL_Wrn,EO_MODBUS,ID,5,'');
					VARS_Alarm:=FALSE;
				END_IF
				(* Next var *)
				VarCnt:=VarCnt+1;
				VarSta:=2;
			ELSE
				IF VarRetry<3 THEN
					VarRetry:=VarRetry+1;
					MB_Start:=TRUE;
				ELSE
					MB_Lock:=FALSE;
					(* Signal error *)
					IF VARS_Alarm=FALSE THEN
						LogEv(EL_Wrn,EO_MODBUS,ID,3,INT_TO_STRING(MB_MASTER.MB_Error));
						VARS_Alarm:=TRUE;
						VarAlarm:=VarCnt-1;
					END_IF
					(* Next var *)
					VarCnt:=VarCnt+1;
					VarSta:=2;
				END_IF
			END_IF
		END_IF

ELSE
	VarSta:=0;
END_CASE
END_ACTION

(* POU Utils Functions/TONOF, ST *)
FUNCTION_BLOCK TONOF
VAR_INPUT
	IN		: BOOL;
	PT_ON	: TIME; (* time to pass, before OUT is set *)
	PT_OF	: TIME; (* time to pass, before OUT is reset *)
END_VAR
VAR_OUTPUT
	OUT		: BOOL;
END_VAR
VAR
	timer	: TON;
END_VAR
IF IN<>OUT THEN
	timer(IN:=TRUE,PT:=SEL(IN,PT_OF,PT_ON));
	IF timer.Q THEN OUT:=IN; END_IF
ELSE
	timer(IN:=FALSE);
END_IF
END_FUNCTION_BLOCK

(* POU Plant_Objects/obj_COMPRESSORE_OLD, ST *)
FUNCTION_BLOCK obj_COMPRESSORE_OLD
VAR CONSTANT

	TimeOutModBus: TON;

END_VAR
VAR_INPUT
	ID			:	BYTE;
	Address		:	BYTE;


	(* Modbus *)
	Refresh_Now	:	BOOL;			(* Richiesta di lettura stato macchina Immediata  *)
	retryErrMax	:	BYTE := 2;

	OnOff		: 	BOOL;

	IndirizzoDaScrivere: WORD;
	DatoDaScrivere: INT;
	ScriviDato: BOOL;
	ScriviCoil: BOOL;

	fWriteAttivazioneComandi:BOOL;


	RUN_REQ: BOOL;
	STOP_REQ:BOOL;
	AgggiornoStartStop: BOOL;

	CARICO_REQ: BOOL;
	RELEASE_REQ: BOOL;
END_VAR
VAR_IN_OUT
	ModBus		:obj_MODBUS;
END_VAR
VAR_OUTPUT
	Run			:	BOOL;

	Status_Log	:	WORD;
	Status_Vis	:	DWORD;
END_VAR
VAR
	(* da diego per gestione stato stringa > 255*)
	temp :STRING(255);
	tempRaw		: ARRAY [0..MAX_SEND_TCP_CLIENT] OF BYTE;
	tempRawLen :DINT;
	longString:STRING(255);

	(* Timer manage switch on/off delay *)
	Delay		: 	TONOF;
	Warning		:	FLT_TAP := (TAP:=100);
	AllarmeCompressore_MB		:	FLT_TAP;
	WarningCompressore_MB		:	FLT_TAP;

	state		:	INT;
	retry		:	BYTE;
	retryErr	:	BYTE;
	ReadTmr		:	TON := (PT:=T#5s);
	fModbusAlr:BOOL;

	Ctrl_Run: BOOL;


	VerificaFuctionCode: INT;
	VerificaNodoLetto: INT;
	ErroreComuModBus: BOOL;
	IndiceErrore: BYTE;

	MB_BitStato: ARRAY [0..1] OF BOOL;
	MB_RegistriLetti: ARRAY [0..1] OF INT;
	MB_RegistriHoldingLetti: ARRAY [0..400] OF INT;
	MB_BitStatoCoil: ARRAY [0..1] OF BOOL;



	AddressRead: BYTE;
	index: BYTE;
	indexErr: BYTE;

	x: INT;
	IndirizzoStart: INT;
	Stop: BOOL;
	start: BOOL;
	StatusControl: ARRAY [0..15] OF BOOL;


END_VAR
(* Call ModBus state machine *)
Stm();

(* Check alarm	*)
CheckAlarm();

(* Seganalzione stato Compressore  *)
IF ErroreComuModBus THEN
		Status_Log:=2; Status_Vis:=16#2020F0;
   ELSIF WarningCompressore_MB.in  THEN
		Status_Log:=1; Status_Vis:=16#20F0F0;
    ELSE
		Status_Log:=0;
		Status_Vis:=16#006000;
END_IF
END_FUNCTION_BLOCK
ACTION AddLogData:
Logger.s1:=INSERT('&COMPINGRML=',BYTE_TO_STRING(ID),11);
IF ID<10 THEN Logger.s1:=INSERT(Logger.s1,'0',11); END_IF

FOR tempRawLen:=0 TO MAX_SEND_TCP_CLIENT DO
                tempRaw[tempRawLen]:=0;
END_FOR

tempRawLen:=0;


temp:=Logger.s1;
ADDSTRING(ADR(tempRaw), ADR(temp), tempRawLen);



temp:=CONCAT(WORD_TO_STRING(Status_Log),';');
ADDSTRING(ADR(tempRaw), ADR(temp), tempRawLen);


(* Sparo gli ingressi Digitali **)
FOR x:= 0 TO 15 DO
	temp:=CONCAT(SEL(StatusControl[x],'0','1'),';');
	ADDSTRING(ADR(tempRaw), ADR(temp), tempRawLen);
END_FOR

(*

temp:=CONCAT(INT_TO_STRING(MB_RegistriHoldingLetti[1]),';');
ADDSTRING(ADR(tempRaw), ADR(temp), tempRawLen);
temp:=CONCAT(INT_TO_STRING(MB_RegistriHoldingLetti[1]),';');
ADDSTRING(ADR(tempRaw), ADR(temp), tempRawLen); *)
temp:=CONCAT(INT_TO_STRING(MB_RegistriHoldingLetti[3]),';');
ADDSTRING(ADR(tempRaw), ADR(temp), tempRawLen);
temp:=CONCAT(INT_TO_STRING(MB_RegistriHoldingLetti[4]),';');
ADDSTRING(ADR(tempRaw), ADR(temp), tempRawLen);
temp:=CONCAT(INT_TO_STRING(MB_RegistriHoldingLetti[5]),';');
ADDSTRING(ADR(tempRaw), ADR(temp), tempRawLen);
temp:=CONCAT(INT_TO_STRING(MB_RegistriHoldingLetti[6]),';');
ADDSTRING(ADR(tempRaw), ADR(temp), tempRawLen);
temp:=CONCAT(INT_TO_STRING(MB_RegistriHoldingLetti[7]),';');
ADDSTRING(ADR(tempRaw), ADR(temp), tempRawLen);
temp:=CONCAT(INT_TO_STRING(MB_RegistriHoldingLetti[8]),';');
ADDSTRING(ADR(tempRaw), ADR(temp), tempRawLen);
temp:=CONCAT(INT_TO_STRING(MB_RegistriHoldingLetti[9]),';');
ADDSTRING(ADR(tempRaw), ADR(temp), tempRawLen);
temp:=CONCAT(INT_TO_STRING(MB_RegistriHoldingLetti[10]),';');
ADDSTRING(ADR(tempRaw), ADR(temp), tempRawLen);
temp:=CONCAT(INT_TO_STRING(MB_RegistriHoldingLetti[20]),';');
ADDSTRING(ADR(tempRaw), ADR(temp), tempRawLen);
temp:=CONCAT(INT_TO_STRING(MB_RegistriHoldingLetti[64]),';');
ADDSTRING(ADR(tempRaw), ADR(temp), tempRawLen);
temp:=CONCAT(INT_TO_STRING(MB_RegistriHoldingLetti[65]),';');
ADDSTRING(ADR(tempRaw), ADR(temp), tempRawLen);
temp:=CONCAT(INT_TO_STRING(MB_RegistriHoldingLetti[66]),';');
ADDSTRING(ADR(tempRaw), ADR(temp), tempRawLen);
temp:=CONCAT(INT_TO_STRING(MB_RegistriHoldingLetti[67]),';');
ADDSTRING(ADR(tempRaw), ADR(temp), tempRawLen);
temp:=CONCAT(INT_TO_STRING(MB_RegistriHoldingLetti[98]),';');
ADDSTRING(ADR(tempRaw), ADR(temp), tempRawLen);
temp:=CONCAT(INT_TO_STRING(MB_RegistriHoldingLetti[103]),';');
ADDSTRING(ADR(tempRaw), ADR(temp), tempRawLen);
temp:=CONCAT(INT_TO_STRING(MB_RegistriHoldingLetti[112]),';');
ADDSTRING(ADR(tempRaw), ADR(temp), tempRawLen);
temp:=CONCAT(INT_TO_STRING(MB_RegistriHoldingLetti[113]),';');
ADDSTRING(ADR(tempRaw), ADR(temp), tempRawLen);
temp:=CONCAT(INT_TO_STRING(MB_RegistriHoldingLetti[114]),';');
ADDSTRING(ADR(tempRaw), ADR(temp), tempRawLen);
temp:=CONCAT(INT_TO_STRING(MB_RegistriHoldingLetti[116]),';');
ADDSTRING(ADR(tempRaw), ADR(temp), tempRawLen);
temp:=CONCAT(INT_TO_STRING(MB_RegistriHoldingLetti[117]),';');
ADDSTRING(ADR(tempRaw), ADR(temp), tempRawLen);
temp:=CONCAT(INT_TO_STRING(MB_RegistriHoldingLetti[123]),';');
ADDSTRING(ADR(tempRaw), ADR(temp), tempRawLen);
temp:=CONCAT(INT_TO_STRING(MB_RegistriHoldingLetti[125]),';');
ADDSTRING(ADR(tempRaw), ADR(temp), tempRawLen);
temp:=CONCAT(INT_TO_STRING(MB_RegistriHoldingLetti[130]),';');
ADDSTRING(ADR(tempRaw), ADR(temp), tempRawLen);
temp:=CONCAT(INT_TO_STRING(MB_RegistriHoldingLetti[255]),';');
ADDSTRING(ADR(tempRaw), ADR(temp), tempRawLen);
temp:=CONCAT(INT_TO_STRING(MB_RegistriHoldingLetti[256]),';');
ADDSTRING(ADR(tempRaw), ADR(temp), tempRawLen);
temp:=CONCAT(INT_TO_STRING(MB_RegistriHoldingLetti[257]),';');
ADDSTRING(ADR(tempRaw), ADR(temp), tempRawLen);
temp:=CONCAT(INT_TO_STRING(MB_RegistriHoldingLetti[258]),';');
ADDSTRING(ADR(tempRaw), ADR(temp), tempRawLen);
temp:=CONCAT(INT_TO_STRING(MB_RegistriHoldingLetti[259]),';');
ADDSTRING(ADR(tempRaw), ADR(temp), tempRawLen);
temp:=CONCAT(INT_TO_STRING(MB_RegistriHoldingLetti[260]),';');
ADDSTRING(ADR(tempRaw), ADR(temp), tempRawLen);
temp:=CONCAT(INT_TO_STRING(MB_RegistriHoldingLetti[261]),';');
ADDSTRING(ADR(tempRaw), ADR(temp), tempRawLen);
temp:=CONCAT(INT_TO_STRING(MB_RegistriHoldingLetti[261]),';');
ADDSTRING(ADR(tempRaw), ADR(temp), tempRawLen);
temp:=CONCAT(INT_TO_STRING(MB_RegistriHoldingLetti[263]),';');
ADDSTRING(ADR(tempRaw), ADR(temp), tempRawLen);
temp:=CONCAT(INT_TO_STRING(MB_RegistriHoldingLetti[264]),';');
ADDSTRING(ADR(tempRaw), ADR(temp), tempRawLen);
temp:=CONCAT(INT_TO_STRING(MB_RegistriHoldingLetti[265]),';');
ADDSTRING(ADR(tempRaw), ADR(temp), tempRawLen);
temp:=CONCAT(INT_TO_STRING(MB_RegistriHoldingLetti[266]),';');
ADDSTRING(ADR(tempRaw), ADR(temp), tempRawLen);
temp:=CONCAT(INT_TO_STRING(MB_RegistriHoldingLetti[267]),';');
ADDSTRING(ADR(tempRaw), ADR(temp), tempRawLen);
temp:=CONCAT(INT_TO_STRING(MB_RegistriHoldingLetti[268]),';');
ADDSTRING(ADR(tempRaw), ADR(temp), tempRawLen);
temp:=CONCAT(INT_TO_STRING(MB_RegistriHoldingLetti[269]),';');
ADDSTRING(ADR(tempRaw), ADR(temp), tempRawLen);
temp:=(INT_TO_STRING(MB_RegistriHoldingLetti[270]));
ADDSTRING(ADR(tempRaw), ADR(temp), tempRawLen);


ADDSTRING(ADR(Logger.TData), ADR(tempRaw), Logger.TLen);
END_ACTION
ACTION CheckAlarm:
(**** GEstione Log ad Evento *****)


	AllarmeCompressore_MB(IN:=MB_RegistriHoldingLetti[1].6 );

	IF AllarmeCompressore_MB.EVH THEN
		LogEv(EL_Alarm,EO_COMPINGRML,ID,1,CONCAT ('AllarmeAttivo_n.', INT_TO_STRING(MB_RegistriHoldingLetti[255])));
	END_IF

	IF AllarmeCompressore_MB.EVL THEN
		LogEv(EL_Log,EO_COMPINGRML,ID,2,CONCAT ('AllarmeRientrato_n.', INT_TO_STRING(MB_RegistriHoldingLetti[255])));
	END_IF


	WarningCompressore_MB(IN:=MB_RegistriHoldingLetti[1].5 );

	IF WarningCompressore_MB.EVH THEN
		LogEv(EL_Wrn,EO_COMPINGRML,ID,1,CONCAT ('AllarmeAttivo_n.', INT_TO_STRING(MB_RegistriHoldingLetti[255])));
	END_IF

	IF WarningCompressore_MB.EVL THEN
		LogEv(EL_Log,EO_COMPINGRML,ID,2,CONCAT ('AllarmeRientrato_n.', INT_TO_STRING(MB_RegistriHoldingLetti[255])));
	END_IF
END_ACTION
ACTION Stm:
CASE state OF
	0:	(* Refresh time manager *)
		ReadTmr(IN:=NOT ReadTmr.Q);
		(*A tempo interrogo il nodo sempre che non ci sia qualcuno che lo sta interrogando in quel momento *)

		IF (ReadTmr.Q AND NodoDaInterrogareCompressoreVecchio=Address )  AND NOT InibiscoModbusCompressoreVecchio THEN
			state := 10;
			ReadTmr.PT := T#100ms;  (* moreno *)
			Refresh_Now := FALSE;
			InibiscoModbusCompressoreVecchio := TRUE;
		END_IF

	(**** Leggo le Analogiche a Disposzione  ****)

	10:	(* richiedo lettura Holding Registere   *)

		Modbus.MB_Query.SlaveAddress := Address;
		Modbus.MB_Query.FunctionCode := 3;
		IndirizzoStart:=1;
		ModBus.MB_Query.Read_StartAddress :=IndirizzoStart - 1 ;
		ModBus.MB_Query.Read_Quantity := 2;
		ModBus.MB_Start := TRUE;
		state := 20;

	20:	(* Risposta all'interrogazione *)
		IF NOT ModBus.MB_Start   THEN
			VerificaFuctionCode:=ModBus.MB_Resp.FunctionCode;
			VerificaNodoLetto:=ModBus.MB_Resp.SlaveAddress;

			IF ModBus.MB_MASTER.MB_Error<>0 THEN
				state := 300;
			ELSE
				FOR x:=0 TO ModBus.MB_Query.Read_Quantity DO
					IF x+IndirizzoStart=3 THEN
						IF  ModBus.MB_Resp.Data[x]<260 THEN    (* condizione perchè questo registro si sporca con un valore 599 *)
				       		MB_RegistriHoldingLetti[x+IndirizzoStart] := ModBus.MB_Resp.Data[x];   	(* Vedi tabella *)
						ELSE
				       		MB_RegistriHoldingLetti[x+IndirizzoStart] := MB_RegistriHoldingLetti[x+IndirizzoStart];   	(* Vedi tabella *)
						END_IF
					ELSE
				       	MB_RegistriHoldingLetti[x+IndirizzoStart] := ModBus.MB_Resp.Data[x];   	(* Vedi tabella *)
					END_IF
				END_FOR

					StatusControl[0]:= MB_RegistriHoldingLetti[IndirizzoStart].0;   	(* Vedi tabella *)
					StatusControl[1]:= MB_RegistriHoldingLetti[IndirizzoStart].1;   	(* Vedi tabella *)
					StatusControl[2]:= MB_RegistriHoldingLetti[IndirizzoStart].2;   	(* Vedi tabella *)
					StatusControl[3]:= MB_RegistriHoldingLetti[IndirizzoStart].3;   	(* Vedi tabella *)
					StatusControl[4]:= MB_RegistriHoldingLetti[IndirizzoStart].4;   	(* Vedi tabella *)
					StatusControl[5]:= MB_RegistriHoldingLetti[IndirizzoStart].5;   	(* Vedi tabella *)
					StatusControl[6]:= MB_RegistriHoldingLetti[IndirizzoStart].6;   	(* Vedi tabella *)
					StatusControl[7]:= MB_RegistriHoldingLetti[IndirizzoStart].7;   	(* Vedi tabella *)
					StatusControl[8]:= MB_RegistriHoldingLetti[IndirizzoStart].8;   	(* Vedi tabella *)
					StatusControl[9]:= MB_RegistriHoldingLetti[IndirizzoStart].9;   	(* Vedi tabella *)
					StatusControl[10]:= MB_RegistriHoldingLetti[IndirizzoStart].10;   	(* Vedi tabella *)
					StatusControl[11]:= MB_RegistriHoldingLetti[IndirizzoStart].11;   	(* Vedi tabella *)
					StatusControl[12]:= MB_RegistriHoldingLetti[IndirizzoStart].12;   	(* Vedi tabella *)
					StatusControl[13]:= MB_RegistriHoldingLetti[IndirizzoStart].13;   	(* Vedi tabella *)
					StatusControl[14]:= MB_RegistriHoldingLetti[IndirizzoStart].14;   	(* Vedi tabella *)
					StatusControl[15]:= MB_RegistriHoldingLetti[IndirizzoStart].15;   	(* Vedi tabella *)






				IndirizzoStart:=3;
				ModBus.MB_Query.Read_StartAddress :=IndirizzoStart-1; 	(* richiedo lettura altri Parametri *)
				ModBus.MB_Query.Read_Quantity := 19;
				ModBus.MB_Start := TRUE;

				state := 40;
			END_IF
		END_IF

	30: (* Rispota Altri paramenti *)
		IF NOT ModBus.MB_Start  THEN

			IF ModBus.MB_MASTER.MB_Error<>0 THEN
				state := 300;
			ELSE

				FOR x:=0 TO ModBus.MB_Query.Read_Quantity DO
					MB_RegistriHoldingLetti[x+IndirizzoStart] := ModBus.MB_Resp.Data[x];   	(* Vedi tabella *)
				END_FOR

				IndirizzoStart:=20;
				ModBus.MB_Query.Read_StartAddress :=IndirizzoStart-1; 	(* richiedo lettura altri Parametri *)
				ModBus.MB_Query.Read_Quantity := 1;
				ModBus.MB_Start := TRUE;

				state := 40;
			END_IF
		END_IF

	40: (* Rispota Altri paramenti *)
		IF NOT ModBus.MB_Start  THEN

			IF ModBus.MB_MASTER.MB_Error<>0 THEN
				state := 300;
			ELSE

				FOR x:=0 TO ModBus.MB_Query.Read_Quantity DO
					MB_RegistriHoldingLetti[x+IndirizzoStart] := ModBus.MB_Resp.Data[x];   	(* Vedi tabella *)
				END_FOR

				IndirizzoStart:=64;
				ModBus.MB_Query.Read_StartAddress :=IndirizzoStart-1; 	(* richiedo lettura altri Parametri *)
				ModBus.MB_Query.Read_Quantity := 4;
				ModBus.MB_Start := TRUE;

				state := 45;
			END_IF
		END_IF

	45: (* Rispota Altri paramenti *)
		IF NOT ModBus.MB_Start  THEN

			IF ModBus.MB_MASTER.MB_Error<>0 THEN
				state := 300;
			ELSE
				FOR x:=0 TO ModBus.MB_Query.Read_Quantity DO
					MB_RegistriHoldingLetti[x+IndirizzoStart] := ModBus.MB_Resp.Data[x];   	(* Vedi tabella *)
				END_FOR

				IndirizzoStart:=96;
				ModBus.MB_Query.Read_StartAddress :=IndirizzoStart-1; 	(* richiedo lettura altri Parametri *)
				ModBus.MB_Query.Read_Quantity := 8;
				ModBus.MB_Start := TRUE;

				state := 50;
			END_IF
		END_IF


	50: (* Rispota Altri paramenti *)
		IF NOT ModBus.MB_Start  THEN

			IF ModBus.MB_MASTER.MB_Error<>0 THEN
				state := 300;
			ELSE
				FOR x:=0 TO ModBus.MB_Query.Read_Quantity DO
					MB_RegistriHoldingLetti[x+IndirizzoStart] := ModBus.MB_Resp.Data[x];   	(* Vedi tabella *)
				END_FOR

				IndirizzoStart:=112;
				ModBus.MB_Query.Read_StartAddress :=IndirizzoStart-1; 	(* richiedo lettura altri Parametri *)
				ModBus.MB_Query.Read_Quantity := 10;
				ModBus.MB_Start := TRUE;


				state := 51;
			END_IF
		END_IF


	51: (* Rispota Altri paramenti *)
		IF NOT ModBus.MB_Start  THEN

			IF ModBus.MB_MASTER.MB_Error<>0 THEN
				state := 300;
			ELSE
				FOR x:=0 TO ModBus.MB_Query.Read_Quantity DO
					MB_RegistriHoldingLetti[x+IndirizzoStart] := ModBus.MB_Resp.Data[x];   	(* Vedi tabella *)
				END_FOR

				IndirizzoStart:=256;
				ModBus.MB_Query.Read_StartAddress :=IndirizzoStart-1; 	(* richiedo lettura altri Parametri *)
				ModBus.MB_Query.Read_Quantity := 14;
				ModBus.MB_Start := TRUE;


				state := 55;
			END_IF
		END_IF


	55: (* Rispota Altri paramenti *)
		IF NOT ModBus.MB_Start  THEN

			IF ModBus.MB_MASTER.MB_Error<>0 THEN
				state := 300;
			ELSE
				FOR x:=0 TO ModBus.MB_Query.Read_Quantity DO
					MB_RegistriHoldingLetti[x+IndirizzoStart] := ModBus.MB_Resp.Data[x];   	(* Vedi tabella *)
				END_FOR

				IndirizzoStart:=122;
				ModBus.MB_Query.Read_StartAddress :=IndirizzoStart-1; 	(* richiedo lettura altri Parametri *)
				ModBus.MB_Query.Read_Quantity := 10;
				ModBus.MB_Start := TRUE;

				state := 56;
			END_IF
		END_IF

	56: (* Rispota Altri paramenti *)
		IF NOT ModBus.MB_Start  THEN

			IF ModBus.MB_MASTER.MB_Error<>0 THEN
				state := 300;
			ELSE
				FOR x:=0 TO ModBus.MB_Query.Read_Quantity DO
					MB_RegistriHoldingLetti[x+IndirizzoStart] := ModBus.MB_Resp.Data[x];   	(* Vedi tabella *)
				END_FOR

				IndirizzoStart:=132;
				ModBus.MB_Query.Read_StartAddress :=IndirizzoStart-1; 	(* richiedo lettura altri Parametri *)
				ModBus.MB_Query.Read_Quantity := 10;
				ModBus.MB_Start := TRUE;

				state := 57;
			END_IF
		END_IF

	57: (* Rispota Altri paramenti *)
		IF NOT ModBus.MB_Start  THEN

			IF ModBus.MB_MASTER.MB_Error<>0 THEN
				state := 300;
			ELSE
				FOR x:=0 TO ModBus.MB_Query.Read_Quantity DO
					MB_RegistriHoldingLetti[x+IndirizzoStart] := ModBus.MB_Resp.Data[x];   	(* Vedi tabella *)
				END_FOR

				IndirizzoStart:=142;
				ModBus.MB_Query.Read_StartAddress :=IndirizzoStart-1; 	(* richiedo lettura altri Parametri *)
				ModBus.MB_Query.Read_Quantity := 10;
				ModBus.MB_Start := TRUE;

				state := 58;
			END_IF
		END_IF

	58: (* Rispota Altri paramenti *)
		IF NOT ModBus.MB_Start  THEN

			IF ModBus.MB_MASTER.MB_Error<>0 THEN
				state := 300;
			ELSE
				FOR x:=0 TO ModBus.MB_Query.Read_Quantity DO
					MB_RegistriHoldingLetti[x+IndirizzoStart] := ModBus.MB_Resp.Data[x];   	(* Vedi tabella *)
				END_FOR

				IndirizzoStart:=250;
				ModBus.MB_Query.Read_StartAddress :=IndirizzoStart-1; 	(* richiedo lettura altri Parametri *)
				ModBus.MB_Query.Read_Quantity := 6;
				ModBus.MB_Start := TRUE;

				state := 60;
			END_IF
		END_IF




	60: (* Rispota Altri paramenti *)
		IF NOT ModBus.MB_Start  THEN

			IF ModBus.MB_MASTER.MB_Error<>0 THEN
				state := 300;
			ELSE
				FOR x:=0 TO ModBus.MB_Query.Read_Quantity DO
					MB_RegistriHoldingLetti[x+IndirizzoStart] := ModBus.MB_Resp.Data[x];   	(* Vedi tabella *)
				END_FOR

				state :=290;
			END_IF
		END_IF


		290:    (* Scrittura il comando di run o stop da remoto*)
		IF NOT ModBus.MB_Start THEN
			IF ModBus.MB_MASTER.MB_Error<>0 THEN (*OR ModBus.MB_MASTER.MB_Error<>0 THEN*)
				state := 300;
			ELSE
				IF AgggiornoStartStop  THEN

					Modbus.MB_Query.FunctionCode := 6;
					Modbus.MB_Query.SlaveAddress := Address;

					IF RUN_REQ THEN
							IndirizzoDaScrivere:=1;
								 DatoDaScrivere:=MB_RegistriHoldingLetti[IndirizzoDaScrivere];
	  							 DatoDaScrivere.0:=TRUE;
  							        DatoDaScrivere.1:=TRUE;
							        DatoDaScrivere.2:=FALSE;
								 RUN_REQ:=FALSE;
					END_IF
					IF STOP_REQ THEN
							IndirizzoDaScrivere:=1;
								 DatoDaScrivere:=MB_RegistriHoldingLetti[IndirizzoDaScrivere];
	  							 DatoDaScrivere.0:=TRUE;
  							        DatoDaScrivere.1:=FALSE;
							        DatoDaScrivere.2:=FALSE;
								STOP_REQ:=FALSE;
					END_IF
					IF RELEASE_REQ THEN
							IndirizzoDaScrivere:=1;
								 DatoDaScrivere:=MB_RegistriHoldingLetti[IndirizzoDaScrivere];
	  							 DatoDaScrivere.0:=FALSE;
  							        DatoDaScrivere.1:=FALSE;
							        DatoDaScrivere.2:=FALSE;
								 RELEASE_REQ:=FALSE;
					END_IF
					IF CARICO_REQ THEN
							IndirizzoDaScrivere:=1;
								 DatoDaScrivere:=MB_RegistriHoldingLetti[IndirizzoDaScrivere];
	  							 DatoDaScrivere.0:=FALSE;
  							        DatoDaScrivere.1:=FALSE;
							        DatoDaScrivere.2:=TRUE;
								 CARICO_REQ:=FALSE;
					END_IF


					ModBus.MB_Query.Write_StartAddress := IndirizzoDaScrivere-1;
					ModBus.MB_Query.Write_Data[0] := DatoDaScrivere;
					ModBus.MB_Start := TRUE;


					AgggiornoStartStop:=FALSE;



					state := 295;
					ELSE
					state := 295;
				END_IF
			END_IF
		END_IF


		295:
		IF NOT ModBus.MB_Start THEN
			IF ModBus.MB_MASTER.MB_Error<>0 THEN (*OR ModBus.MB_MASTER.MB_Error<>0 THEN*)
				state := 300;
			ELSE
				IF fModbusAlr THEN fModbusAlr := FALSE; END_IF
				NodoDaInterrogareCompressoreVecchio:=Address+1;
				InibiscoModbusCompressoreVecchio:=FALSE;
				retryErr := 0;
				retry := 0;
				state := 0;
					IF fModbusAlr=FALSE AND ErroreComuModBus=TRUE THEN
						LogEv(EL_Log,EO_COMPINGRR,ID,62,'ComunicazioneModBus_OK');
						ErroreComuModBus := FALSE;
				(*	WarningCtr := SEL(WarningCtr=0, WarningCtr-1, 0); *)
					END_IF


			END_IF
		END_IF



	(**** CHECK MODBUS ERROR ****)
	300: 	(* Release MODBUS *)
			InibiscoModbusCompressoreVecchio:=FALSE;
			(* Retries *)
			retry:=retry+1;
			IF retry>3 THEN
				retry:=0;

				(* Verify if slave is dead *)
				IF retryErr < retryErrMaX THEN
					retryErr := retryErr + 1;
				ELSE
					fModbusAlr := TRUE;
					(* Verify ModBus error	*)

					IF fModbusAlr AND ErroreComuModBus=FALSE THEN
						LogEv(EL_Alarm,EO_COMPINGRR,ID,61,CONCAT('ErroreModbus_',INT_TO_STRING(ModBus.MB_MASTER.MB_Error)));
						ErroreComuModBus := TRUE;
					END_IF
				END_IF

				END_IF
			Refresh_Now := FALSE;
			NodoDaInterrogareCompressoreVecchio:=Address+1;
			state:=0;
END_CASE




(* Controllo Time Out Ciclo ModBus *)

TimeOutModBus(In:=state<>0,PT:=t#3s);
IF TimeOutModBus.Q THEN
	State:=0;
	Refresh_Now:=TRUE;  (* Rilancio la lettura del nodo *)
	IF MODBUS.MB_Lock=TRUE THEN MODBUS.MB_Lock:=FALSE;END_IF
	IF InibiscoModbusCompressoreVecchio=TRUE THEN InibiscoModbusCompressoreVecchio:=FALSE;END_IF
	NodoDaInterrogareCompressoreVecchio:=Address+1;

END_IF
END_ACTION

(* POU Plant_Objects/obj_ESSICATORE, ST *)
FUNCTION_BLOCK obj_ESSICATORE
VAR CONSTANT

	TimeOutModBus: TON;


END_VAR
VAR_INPUT
	ID			:	BYTE;
	Address		:	BYTE;


	(* Modbus *)
	Refresh_Now	:	BOOL;			(* Richiesta di lettura stato macchina Immediata  *)
	retryErrMax	:	BYTE := 2;

	OnOff		: 	BOOL;

	IndirizzoDaScrivere: WORD;
	DatoDaScrivere: INT;
	ScriviDato: BOOL;
	ScriviCoil: BOOL;

	fWriteAttivazioneComandi:BOOL;

	RUN_REQ: BOOL;
	STOP_REQ:BOOL;
	AgggiornoStartStop: BOOL;
END_VAR
VAR_IN_OUT
	ModBus		:obj_MODBUS_Free;
END_VAR
VAR_OUTPUT
	Run			:	BOOL;

	Status_Log	:	WORD;
	Status_Vis	:	DWORD;
END_VAR
VAR
	(* da diego per gestione stato stringa > 255*)
	temp :STRING(255);
	tempRaw		: ARRAY [0..MAX_SEND_TCP_CLIENT] OF BYTE;
	tempRawLen :DINT;
	longString:STRING(255);

	(* Timer manage switch on/off delay *)
	Delay		: 	TONOF;
	Warning		:	FLT_TAP := (TAP:=100);
	AllarmeCompressore_MB		:	FLT_TAP;

	state		:	INT;
	retry		:	BYTE;
	retryErr	:	BYTE;
	ReadTmr		:	TON := (PT:=T#5s);
	fModbusAlr:BOOL;

	Ctrl_Run: BOOL;


	VerificaFuctionCode: INT;
	VerificaNodoLetto: INT;
	ErroreComuModBus: BOOL;
	IndiceErrore: BYTE;

	MB_BitStato: ARRAY [0..1] OF BOOL;
	MB_RegistriLetti: ARRAY [0..1] OF INT;
	MB_RegistriHoldingLetti: ARRAY [0..500] OF INT;
	MB_BitStatoCoil: ARRAY [0..1] OF BOOL;



	AddressRead: BYTE;
	index: BYTE;
	indexErr: BYTE;





	x: INT;
	moreno1: INT;
	moreno2: INT;
	IndirizzoStart: INT;

	Parametro1280: WORD;
	Parametro1282: WORD;
	morenoind: INT;
	morenoqta: INT;
	Probe1: INT;
	StatusProbe1: INT;
	Probe2: INT;
	StatusProbe2: INT;
	Probe3: INT;
	StatusProbe3: INT;
	Probe4: INT;
	StatusProbe4: INT;
	TempoPausa: TON;
END_VAR
(* Call ModBus state machine *)
Stm();

(* Check alarm	*)

(* Seganalzione stato Compressore  *)
IF ErroreComuModBus THEN
		Status_Log:=2; Status_Vis:=16#2020F0;
(*	ELSIF Warning OR Warning2 THEN
		Status_Log:=1; Status_Vis:=16#20F0F0; *)
    ELSE
		Status_Log:=0;
		Status_Vis:=16#006000;
END_IF
END_FUNCTION_BLOCK
ACTION AddLogData:
Logger.s1:=CONCAT('&','ESC');
IF ID<10 THEN Logger.s1:=CONCAT(Logger.s1,'0');END_IF
Logger.s1:=CONCAT(Logger.s1,BYTE_TO_STRING(ID));
Logger.s1:=CONCAT(Logger.s1,'=');


FOR tempRawLen:=0 TO MAX_SEND_TCP_CLIENT DO
                tempRaw[tempRawLen]:=0;
END_FOR

tempRawLen:=0;


temp:=Logger.s1;
ADDSTRING(ADR(tempRaw), ADR(temp), tempRawLen);

temp:=CONCAT(WORD_TO_STRING(Status_Log),';');
ADDSTRING(ADR(tempRaw), ADR(temp), tempRawLen);
temp:=(INT_TO_STRING(Probe1));
ADDSTRING(ADR(tempRaw), ADR(temp), tempRawLen);


ADDSTRING(ADR(Logger.TData), ADR(tempRaw), Logger.TLen);
END_ACTION
ACTION Stm:
CASE state OF
	0:	(* Refresh time manager *)
		ReadTmr(IN:=NOT ReadTmr.Q);
		(*A tempo interrogo il nodo sempre che non ci sia qualcuno che lo sta interrogando in quel momento *)

		IF (ReadTmr.Q AND NodoDaInterrogareEssicatore=Address ) OR Refresh_Now AND NOT InibiscoModbusEssicatore THEN
			state := 10;
			ReadTmr.PT := T#3000ms;  (* moreno *)
			Refresh_Now := FALSE;
			InibiscoModbusEssicatore := TRUE;
			TempoPausa(IN:=FALSE , PT:=t#200ms , Q=> , ET=> );

		END_IF

	(**** Leggo le Analogiche a Disposzione  ****)

	10:	(* richiedo lettura Holding Registere   *)


		Modbus.MB_MASTER.cbsCOM_BYTESIZE:=BS_8;
		Modbus.MB_MASTER.cpCOM_PARITY:=PARITY_NO;

		Modbus.MB_Query.SlaveAddress := Address;
		Modbus.MB_Query.FunctionCode := 3;
		IndirizzoStart:=257;
		ModBus.MB_Query.Read_StartAddress :=IndirizzoStart-1  ;
		ModBus.MB_Query.Read_Quantity := 2;(*19;*)
		state := 17;

	17: TempoPausa(IN:=TRUE , PT:=t#100ms , Q=> , ET=> );
			IF TempoPausa.Q THEN
				ModBus.MB_Start := TRUE;
				TempoPausa(IN:=FALSE , PT:=t#200ms , Q=> , ET=> );
				state := state+1;;
			END_IF


	18:	(* Risposta all'interrogazione *)
		IF NOT ModBus.MB_Start   THEN
			VerificaFuctionCode:=ModBus.MB_Resp.FunctionCode;
			VerificaNodoLetto:=ModBus.MB_Resp.SlaveAddress;

			IF ModBus.MB_MASTER.MB_Error=0 THEN
				Probe1:=ModBus.MB_Resp.Data[0];
				StatusProbe1:=ModBus.MB_Resp.Data[1];
			END_IF

				IndirizzoStart:=259;
				ModBus.MB_Query.Read_StartAddress :=IndirizzoStart - 1 ;
				ModBus.MB_Query.Read_Quantity :=2;
				state :=19;
			END_IF

	19: TempoPausa(IN:=TRUE , PT:=t#500ms , Q=> , ET=> );
			IF TempoPausa.Q THEN
			ModBus.MB_Start := TRUE;
			TempoPausa(IN:=FALSE , PT:=t#200ms , Q=> , ET=> );
				state := state+1;;
			END_IF

	20:	(* Risposta all'interrogazione *)
		IF NOT ModBus.MB_Start   THEN
			VerificaFuctionCode:=ModBus.MB_Resp.FunctionCode;
			VerificaNodoLetto:=ModBus.MB_Resp.SlaveAddress;

			IF ModBus.MB_MASTER.MB_Error=0 THEN
				Probe2:=ModBus.MB_Resp.Data[0];
				StatusProbe2:=ModBus.MB_Resp.Data[1];
			END_IF

				IndirizzoStart:=261;
				ModBus.MB_Query.Read_StartAddress :=IndirizzoStart - 1 ;
				ModBus.MB_Query.Read_Quantity :=2;

				state := 29;
		END_IF
	29: TempoPausa(IN:=TRUE , PT:=t#500ms , Q=> , ET=> );
			IF TempoPausa.Q THEN
				ModBus.MB_Start := TRUE;
				TempoPausa(IN:=FALSE , PT:=t#200ms , Q=> , ET=> );
				state := state+1;;
			END_IF
	30: (* Rispota Altri paramenti *)
		IF NOT ModBus.MB_Start  THEN

			IF ModBus.MB_MASTER.MB_Error=0 THEN
				Probe3:=ModBus.MB_Resp.Data[0];
				StatusProbe3:=ModBus.MB_Resp.Data[1];
			END_IF



				IndirizzoStart:=263;
				ModBus.MB_Query.Read_StartAddress :=IndirizzoStart - 1 ;
				ModBus.MB_Query.Read_Quantity := 1;

				state := 34;
			END_IF

	34: TempoPausa(IN:=TRUE , PT:=t#500ms , Q=> , ET=> );
			IF TempoPausa.Q THEN
				ModBus.MB_Start := TRUE;
				TempoPausa(IN:=FALSE , PT:=t#200ms , Q=> , ET=> );
				state := state+1;;
			END_IF

	35: (* Rispota Altri paramenti *)
		IF NOT ModBus.MB_Start  THEN

			IF ModBus.MB_MASTER.MB_Error=0 THEN
				Probe4:=ModBus.MB_Resp.Data[0];
				StatusProbe4:=ModBus.MB_Resp.Data[1];
			END_IF


				state := 295;
		END_IF

	39: TempoPausa(IN:=TRUE , PT:=t#500ms , Q=> , ET=> );
			IF TempoPausa.Q THEN
				ModBus.MB_Start := TRUE;
				TempoPausa(IN:=FALSE , PT:=t#200ms , Q=> , ET=> );
				state := state+1;;
			END_IF
	40: (* Rispota Altri paramenti *)
		IF NOT ModBus.MB_Start  THEN

			IF ModBus.MB_MASTER.MB_Error<>0 THEN
				state := 300;
			ELSE

(*				FOR x:=0 TO ModBus.MB_Query.Read_Quantity DO
					MB_RegistriHoldingLetti[x+IndirizzoStart] := ModBus.MB_Resp.Data[x];   	(* Vedi tabella *)
				END_FOR *)


				Probe4:=ModBus.MB_Resp.Data[0];
				StatusProbe4:=ModBus.MB_Resp.Data[1];


				state := 295;
			END_IF
		END_IF

	45: (* Rispota Altri paramenti *)
		IF NOT ModBus.MB_Start  THEN

			IF ModBus.MB_MASTER.MB_Error<>0 THEN
				state := 300;
			ELSE
				FOR x:=0 TO ModBus.MB_Query.Read_Quantity DO
					MB_RegistriHoldingLetti[x+IndirizzoStart] := ModBus.MB_Resp.Data[x];   	(* Vedi tabella *)
				END_FOR
				Parametro1282:= ModBus.MB_Resp.Data[0];


		(*		IndirizzoStart:=110;
				ModBus.MB_Query.Read_StartAddress :=IndirizzoStart - 1 ;
				ModBus.MB_Query.Read_Quantity := 19;
				ModBus.MB_Start := TRUE;    *)

				state := 295;
			END_IF
		END_IF


	50: (* Rispota Altri paramenti *)
		IF NOT ModBus.MB_Start  THEN

			IF ModBus.MB_MASTER.MB_Error<>0 THEN
				state := 300;
			ELSE
				FOR x:=0 TO ModBus.MB_Query.Read_Quantity DO
					MB_RegistriHoldingLetti[x+IndirizzoStart] := ModBus.MB_Resp.Data[x];   	(* Vedi tabella *)
				END_FOR

				IndirizzoStart:=130;
				ModBus.MB_Query.Read_StartAddress :=IndirizzoStart - 1 ;
				ModBus.MB_Query.Read_Quantity := 5;
				ModBus.MB_Start := TRUE;


				state := 55;
			END_IF
		END_IF

	55: (* Rispota Altri paramenti *)
		IF NOT ModBus.MB_Start  THEN

			IF ModBus.MB_MASTER.MB_Error<>0 THEN
				state := 300;
			ELSE
				FOR x:=0 TO ModBus.MB_Query.Read_Quantity DO
					MB_RegistriHoldingLetti[x+IndirizzoStart] := ModBus.MB_Resp.Data[x];   	(* Vedi tabella *)
				END_FOR

				IndirizzoStart:=240;
				ModBus.MB_Query.Read_StartAddress :=IndirizzoStart - 1 ;
				ModBus.MB_Query.Read_Quantity := 3;
				ModBus.MB_Start := TRUE;

				state := 60;
			END_IF
		END_IF

	60: (* Rispota Altri paramenti *)
		IF NOT ModBus.MB_Start  THEN

			IF ModBus.MB_MASTER.MB_Error<>0 THEN
				state := 300;
			ELSE
				FOR x:=0 TO ModBus.MB_Query.Read_Quantity DO
					MB_RegistriHoldingLetti[x+IndirizzoStart] := ModBus.MB_Resp.Data[x];   	(* Vedi tabella *)
				END_FOR

				state :=290;
			END_IF
		END_IF


		290:    (* Scrittura il comando di run o stop da remoto*)
		IF NOT ModBus.MB_Start THEN
			IF ModBus.MB_MASTER.MB_Error<>0 THEN (*OR ModBus.MB_MASTER.MB_Error<>0 THEN*)
				state := 300;
			ELSE
				IF AgggiornoStartStop  THEN

					Modbus.MB_Query.FunctionCode := 6;
					Modbus.MB_Query.SlaveAddress := Address;
					ModBus.MB_Query.Write_StartAddress := IndirizzoDaScrivere-1;
					ModBus.MB_Query.Write_Quantity :=1;


					 DatoDaScrivere:=MB_RegistriHoldingLetti[IndirizzoDaScrivere];
	  				 DatoDaScrivere.0:=FALSE;

					IF RUN_REQ THEN
								 DatoDaScrivere:=MB_RegistriHoldingLetti[IndirizzoDaScrivere];
	  							 DatoDaScrivere.0:=TRUE;
  							        DatoDaScrivere.1:=TRUE;
					END_IF
					IF STOP_REQ THEN
								 DatoDaScrivere:=MB_RegistriHoldingLetti[IndirizzoDaScrivere];
	  							 DatoDaScrivere.0:=TRUE;
  							        DatoDaScrivere.1:=FALSE;
					END_IF


					ModBus.MB_Query.Write_Data[0] := DatoDaScrivere;
					ModBus.MB_Start := TRUE;
					state := 291;
					AgggiornoStartStop:=FALSE;
				ELSE
					state := 291;
				END_IF
			END_IF
		END_IF
		291:    (* Scrittura BOOL - COIL o WORD *)
		IF NOT ModBus.MB_Start THEN
			IF ModBus.MB_MASTER.MB_Error<>0 THEN (*OR ModBus.MB_MASTER.MB_Error<>0 THEN*)
				state := 300;
			ELSE
				IF ScriviDato THEN
					IF ScriviCoil THEN
						Modbus.MB_Query.FunctionCode := 5;
					ELSE
						Modbus.MB_Query.FunctionCode := 6;
					END_IF
					Modbus.MB_Query.SlaveAddress := Address;
					ModBus.MB_Query.Write_StartAddress := IndirizzoDaScrivere-1;
					ModBus.MB_Query.Write_Quantity :=1;
					ModBus.MB_Query.Write_Data[0] := DatoDaScrivere;
					ModBus.MB_Start := TRUE;
						IF ScriviCoil THEN
							IF 	MB_BitStato[IndirizzoDaScrivere]=WORD_TO_BOOL(DatoDaScrivere-1) THEN
								ScriviDato:=FALSE;
							END_IF
						ELSE
							IF 	MB_RegistriHoldingLetti[IndirizzoDaScrivere]=DatoDaScrivere THEN
								ScriviDato:=FALSE;
							END_IF
						END_IF
					state := 295;
				ELSE
					state := 295;
				END_IF
			END_IF
		END_IF




		295:
		IF NOT ModBus.MB_Start THEN
			IF ModBus.MB_MASTER.MB_Error<>0 THEN (*OR ModBus.MB_MASTER.MB_Error<>0 THEN*)
				state := 300;
			ELSE
				IF fModbusAlr THEN fModbusAlr := FALSE; END_IF
				NodoDaInterrogareEssicatore:=Address+1;
				InibiscoModbusEssicatore:=FALSE;
				retryErr := 0;
				retry := 0;
				state := 0;
					IF fModbusAlr=FALSE AND ErroreComuModBus=TRUE THEN
						LogEv(EL_Log,EO_COMPINGRML,ID,62,'ComunicazioneModBus_OK');
						ErroreComuModBus := FALSE;
				(*	WarningCtr := SEL(WarningCtr=0, WarningCtr-1, 0); *)
					END_IF
			END_IF


		END_IF




	(**** CHECK MODBUS ERROR ****)
	300: 	(* Release MODBUS *)
			InibiscoModbusEssicatore:=FALSE;
			(* Retries *)
			retry:=retry+1;
			IF retry>3 THEN
				retry:=0;

				(* Verify if slave is dead *)
				IF retryErr < retryErrMaX THEN
					retryErr := retryErr + 1;
				ELSE
					fModbusAlr := TRUE;
					(* Verify ModBus error	*)

					IF fModbusAlr AND ErroreComuModBus=FALSE THEN
						LogEv(EL_Alarm,EO_COMPINGRML,ID,61,CONCAT('ErroreModbus_',INT_TO_STRING(ModBus.MB_MASTER.MB_Error)));
						ErroreComuModBus := TRUE;
					END_IF
				END_IF

				END_IF
			Refresh_Now := FALSE;
			NodoDaInterrogareEssicatore:=Address+1;
			state:=0;
END_CASE




(* Controllo Time Out Ciclo ModBus *)

TimeOutModBus(In:=state<>0,PT:=t#30s);
IF TimeOutModBus.Q THEN
	State:=0;
	Refresh_Now:=TRUE;  (* Rilancio la lettura del nodo *)
	IF MODBUS.MB_Lock=TRUE THEN MODBUS.MB_Lock:=FALSE;END_IF
	IF InibiscoModbusEssicatore=TRUE THEN InibiscoModbusEssicatore:=FALSE;END_IF
	NodoDaInterrogareEssicatore:=Address+1;

END_IF
END_ACTION

(* POU obj_MODBUS_Free, ST *)
FUNCTION_BLOCK obj_MODBUS_Free
(* === MODBUS PROTOCOL INTERFACE ===
   v1.1[19/06/15] - Added new VARS allocation and searching
*)
VAR CONSTANT
	VARS_Max	: BYTE := 32;
END_VAR
VAR_INPUT
	(* Settings *)
	ID			: BYTE;
	COM			: BYTE;
	BAUDRATE	: COM_BAUDRATE;
	RS485		: BOOL := FALSE;

	N_STOPBits	:BYTE:=1;

 	(* Interface *)
	MB_MASTER	: MODBUS_EXTENDED_MASTER;
	MB_Start	: BOOL;
	MB_Query	: typModbusExtendedQuery;
	MB_Resp		: typModbusResponse;
	MB_Lock		: BOOL;
	MB_timeOut	: TIME := t#500ms;

	(* Variables management *)
	VARS_En		: BOOL;
	VARS		: ARRAY [0..VARS_Max] OF typ_MODBUS_VAR;
	VARS_Check	: BOOL;
	VARS_Alarm	: BOOL;

	(* Variables allocation *)
	VAR_Pointer : POINTER TO ARRAY[0..99] OF WORD;
	VAR_Cfg		: POINTER TO typ_MODBUS_VAR;
END_VAR
VAR_OUTPUT
	(* Status *)
	Status_Log	: BYTE;
	Status_Vis	: DWORD;
END_VAR
VAR
	sta         : BYTE :=0;
	i			: BYTE;
	j			: BYTE;
	Alarm		: FLT_EVENT;
	
	VarTmr		: TON := (PT:=T#1s);
	VarSta		: BYTE; (* Status *)
	VarCnt		: BYTE; (* Scan counter *)
	VarRetry	: BYTE;
	VarAlarm	: BYTE; (* Last variable with errors *)
END_VAR
IF N_STOPBits=1 THEN MB_MASTER.csCOM_STOPBITS:=STOPBITS_1;END_IF
IF N_STOPBits=2 THEN MB_MASTER.csCOM_STOPBITS:=STOPBITS_2;END_IF

MB_MASTER(ENABLE:=TRUE,	ASCII_Mode:=FALSE, bCOM_PORT:=COM, cbCOM_BAUDRATE:=BAUDRATE,
		cfCOM_FLOW_CONTROL:=SEL(RS485,NO_FLOW_CONTROL,HALFDUPLEX),
		tTIME_OUT:=MB_timeOut,	StartFunction:=MB_Start, ExtQuery:=MB_Query, Response:=MB_Resp);

(* Process variable management *)
IF VARS_En THEN VARS_Process(); END_IF

(* Check status *)
Alarm(IN:=(MB_MASTER.bInterfaceError<>0));
IF Alarm.EVH THEN
	LogEv(SEL(MB_MASTER.bInterfaceError<>3,EL_Wrn,EL_Alarm),EO_MODBUS,ID,1,BYTE_TO_STRING(MB_MASTER.bInterfaceError));
END_IF
IF Alarm.EVL THEN								(* Trigger a fall edge: MODBUS back working *)
	LogEv(EL_Log,EO_MODBUS,ID,2,'MODBUS_OK');
END_IF

